(* Logix 5000 project; controller reports 1756-L63 rev 20.11; software revision 20.04; part 47 of 52 *)

        [152].log_data[58].time := 3600.0, [152].log_data[58].valid := 1, [152].log_data[59].time := 3600.0, [152].log_data[59].valid := 1, [152].log_data[60].valid := 1, [152].log_data[61].valid := 1, [152].log_data[62].valid := 1, [152].log_data[63].valid := 1, [152].log_data[64].valid := 1, [152].log_data[65].valid := 1, [152].log_data[66].valid := 1, [152].log_data[67].valid := 1, [152].log_data[68].valid := 1, [152].log_data[69].valid := 1, [152].log_data[70].valid := 1, [152].log_data[71].valid := 1, [152].log_data[72].valid := 1, [152].log_data[73].valid := 1, [152].log_data[74].valid := 1, [152].log_data[75].valid := 1, [152].log_data[76].valid := 1, [152].log_data[77].valid := 1, [152].log_data[78].valid := 1, [152].log_data[79].valid := 1, [152].log_data[80].valid := 1, [152].log_data[81].valid := 1, [152].log_data[82].valid := 1, [152].log_data[83].valid := 1, [152].log_data[84].valid := 1, [152].log_data[85].valid := 1, [152].log_data[86].valid := 1, [152].log_data[87].valid := 1, [152].log_data[88].valid := 1, [152].log_data[89].valid := 1, [152].log_data[90].valid := 1, [152].log_data[91].valid := 1, [152].log_data[92].valid := 1, [152].log_data[93].valid := 1, [152].log_data[94].valid := 1, [152].log_data[95].valid := 1, [152].log_data[96].valid := 1, [152].log_data[97].valid := 1, [152].log_data[98].valid := 1, [152].log_data[99].valid := 1, [152].log_data[100].valid := 1, [152].log_data[101].valid := 1, [152].log_data[102].valid := 1, [152].log_data[103].valid := 1, [152].log_data[104].valid := 1, [152].log_data[105].valid := 1, [152].log_data[106].valid := 1, [152].log_data[107].valid := 1, [152].log_data[108].valid := 1, [152].log_data[109].valid := 1, [152].log_data[110].valid := 1, [152].log_data[111].valid := 1, [152].log_data[112].valid := 1, [152].log_data[113].valid := 1, [152].log_data[114].valid := 1, [152].log_data[115].valid := 1,
        [152].log_data[116].valid := 1, [152].log_data[117].valid := 1, [152].log_data[118].valid := 1, [152].log_data[119].valid := 1, [152].log_data[120].valid := 1, [152].log_data[121].valid := 1, [152].log_data[122].valid := 1, [152].log_data[123].valid := 1, [152].log_data[124].valid := 1, [152].time.Year := 2023, [152].time.Month := 1, [152].time.Day := 19, [152].time.Hour := 11, [152].time.Minute := 59, [152].time.Second := 59, [153].log_data[0].min := 1.0, [153].log_data[0].max := 1.0, [153].log_data[0].total := 3600.0, [153].log_data[0].time := 3600.0, [153].log_data[0].valid := 1, [153].log_data[1].time := 3600.0, [153].log_data[1].valid := 1, [153].log_data[2].time := 3600.0, [153].log_data[2].valid := 1, [153].log_data[3].time := 3600.0, [153].log_data[3].valid := 1, [153].log_data[4].time := 3600.0, [153].log_data[4].valid := 1, [153].log_data[5].time := 3600.0, [153].log_data[5].valid := 1, [153].log_data[6].time := 3600.0, [153].log_data[6].valid := 1, [153].log_data[7].time := 3600.0, [153].log_data[7].valid := 1, [153].log_data[8].min := 1.0, [153].log_data[8].max := 1.0, [153].log_data[8].total := 3600.0, [153].log_data[8].time := 3600.0, [153].log_data[8].valid := 1, [153].log_data[9].min := 1.0, [153].log_data[9].max := 1.0, [153].log_data[9].total := 3600.0, [153].log_data[9].time := 3600.0, [153].log_data[9].valid := 1, [153].log_data[10].min := 1.0, [153].log_data[10].max := 1.0, [153].log_data[10].total := 3600.0, [153].log_data[10].time := 3600.0, [153].log_data[10].valid := 1, [153].log_data[11].time := 3600.0, [153].log_data[11].valid := 1, [153].log_data[12].min := 1.0, [153].log_data[12].max := 1.0, [153].log_data[12].total := 3600.0, [153].log_data[12].time := 3600.0, [153].log_data[12].valid := 1, [153].log_data[13].min := 1.0, [153].log_data[13].max := 1.0, [153].log_data[13].total := 3600.0, [153].log_data[13].time := 3600.0,
        [153].log_data[13].valid := 1, [153].log_data[14].time := 3600.0, [153].log_data[14].valid := 1, [153].log_data[15].time := 3600.0, [153].log_data[15].valid := 1, [153].log_data[16].time := 3600.0, [153].log_data[16].valid := 1, [153].log_data[17].min := 1.0, [153].log_data[17].max := 1.0, [153].log_data[17].total := 3600.0, [153].log_data[17].time := 3600.0, [153].log_data[17].valid := 1, [153].log_data[18].time := 3600.0, [153].log_data[18].valid := 1, [153].log_data[19].time := 3600.0, [153].log_data[19].valid := 1, [153].log_data[20].time := 3600.0, [153].log_data[20].valid := 1, [153].log_data[21].min := 1.0, [153].log_data[21].max := 1.0, [153].log_data[21].total := 3600.0, [153].log_data[21].time := 3600.0, [153].log_data[21].valid := 1, [153].log_data[22].time := 3600.0, [153].log_data[22].valid := 1, [153].log_data[23].time := 3600.0, [153].log_data[23].valid := 1, [153].log_data[24].time := 3600.0, [153].log_data[24].valid := 1, [153].log_data[25].time := 3600.0, [153].log_data[25].valid := 1, [153].log_data[26].time := 3600.0, [153].log_data[26].valid := 1, [153].log_data[27].time := 3600.0, [153].log_data[27].valid := 1, [153].log_data[28].time := 3600.0, [153].log_data[28].valid := 1, [153].log_data[29].min := 1.0, [153].log_data[29].max := 1.0, [153].log_data[29].total := 3600.0, [153].log_data[29].time := 3600.0, [153].log_data[29].valid := 1, [153].log_data[30].min := 1.0, [153].log_data[30].max := 1.0, [153].log_data[30].total := 3600.0, [153].log_data[30].time := 3600.0, [153].log_data[30].valid := 1, [153].log_data[31].max := 1.0, [153].log_data[31].total := 1629.749, [153].log_data[31].time := 3600.0, [153].log_data[31].valid := 1, [153].log_data[32].max := 1.0, [153].log_data[32].total := 1481.7471, [153].log_data[32].time := 3600.0, [153].log_data[32].maxminute := 11, [153].log_data[32].valid := 1, [153].log_data[33].time := 3600.0, [153].log_data[33].valid := 1, [153].log_data[34].time := 3600.0, [153].log_data[34].valid := 1,
        [153].log_data[35].max := 1.0, [153].log_data[35].total := 1629.998, [153].log_data[35].time := 3600.0, [153].log_data[35].maxminute := 8, [153].log_data[35].valid := 1, [153].log_data[36].max := 1.0, [153].log_data[36].total := 1480.249, [153].log_data[36].time := 3600.0, [153].log_data[36].minminute := 6, [153].log_data[36].valid := 1, [153].log_data[37].time := 3600.0, [153].log_data[37].valid := 1, [153].log_data[38].time := 3600.0, [153].log_data[38].valid := 1, [153].log_data[39].min := 0.9945885, [153].log_data[39].max := 1.0051882, [153].log_data[39].total := 3601.9607, [153].log_data[39].time := 3600.0, [153].log_data[39].minminute := 59, [153].log_data[39].maxminute := 44, [153].log_data[39].valid := 1, [153].log_data[40].min := 7.5950956, [153].log_data[40].max := 7.6195536, [153].log_data[40].total := 27406.98, [153].log_data[40].time := 3600.0, [153].log_data[40].minminute := 52, [153].log_data[40].maxminute := 59, [153].log_data[40].valid := 1, [153].log_data[41].min := 0.021362305, [153].log_data[41].max := 0.023521485, [153].log_data[41].total := 80.782776, [153].log_data[41].time := 3600.0, [153].log_data[41].minminute := 25, [153].log_data[41].maxminute := 24, [153].log_data[41].valid := 1, [153].log_data[42].min := 2.290936, [153].log_data[42].max := 2.296236, [153].log_data[42].total := 8256.996, [153].log_data[42].time := 3600.0, [153].log_data[42].minminute := 43, [153].log_data[42].maxminute := 14, [153].log_data[42].valid := 1, [153].log_data[43].min := -0.27999878, [153].log_data[43].max := -0.22000122, [153].log_data[43].total := -891.35376, [153].log_data[43].time := 3600.0, [153].log_data[43].maxminute := 45, [153].log_data[43].valid := 1, [153].log_data[44].min := -0.30000305, [153].log_data[44].max := -0.26000214, [153].log_data[44].total := -1000.0248, [153].log_data[44].time := 3600.0, [153].log_data[44].maxminute := 35, [153].log_data[44].valid := 1, [153].log_data[45].time := 3600.0, [153].log_data[45].valid := 1, [153].log_data[46].time := 3600.0, [153].log_data[46].valid := 1, [153].log_data[47].time := 3600.0, [153].log_data[47].valid := 1,
        [153].log_data[48].min := 6.567313, [153].log_data[48].max := 6.784686, [153].log_data[48].total := 24147.303, [153].log_data[48].time := 3600.0, [153].log_data[48].minminute := 14, [153].log_data[48].maxminute := 29, [153].log_data[48].valid := 1, [153].log_data[49].min := 6.8652577, [153].log_data[49].max := 9.493403, [153].log_data[49].total := 29615.246, [153].log_data[49].time := 3600.0, [153].log_data[49].minminute := 15, [153].log_data[49].maxminute := 59, [153].log_data[49].valid := 1, [153].log_data[50].min := 2.0285335, [153].log_data[50].max := 2.1149805, [153].log_data[50].total := 7461.926, [153].log_data[50].time := 3600.0, [153].log_data[50].minminute := 58, [153].log_data[50].valid := 1, [153].log_data[51].time := 3600.0, [153].log_data[51].valid := 1, [153].log_data[52].min := -2.7600021, [153].log_data[52].max := 0.13999939, [153].log_data[52].total := -7610.8003, [153].log_data[52].time := 3600.0, [153].log_data[52].minminute := 21, [153].log_data[52].maxminute := 31, [153].log_data[52].valid := 1, [153].log_data[53].min := -2.5, [153].log_data[53].max := 0.27999878, [153].log_data[53].total := -7005.6523, [153].log_data[53].time := 3600.0, [153].log_data[53].minminute := 50, [153].log_data[53].maxminute := 7, [153].log_data[53].valid := 1, [153].log_data[54].max := 0.5255, [153].log_data[54].total := 1233.0619, [153].log_data[54].time := 3600.0, [153].log_data[54].valid := 1, [153].log_data[55].max := 0.55300003, [153].log_data[55].total := 1235.2316, [153].log_data[55].time := 3600.0, [153].log_data[55].minminute := 6, [153].log_data[55].maxminute := 50, [153].log_data[55].valid := 1, [153].log_data[56].min := 0.15895009, [153].log_data[56].max := 0.15946046, [153].log_data[56].total := 573.08417, [153].log_data[56].time := 3600.0, [153].log_data[56].minminute := 2, [153].log_data[56].maxminute := 44, [153].log_data[56].valid := 1, [153].log_data[57].min := 0.18721606, [153].log_data[57].max := 0.18976782, [153].log_data[57].total := 676.8789, [153].log_data[57].time := 3600.0, [153].log_data[57].minminute := 24, [153].log_data[57].maxminute := 6, [153].log_data[57].valid := 1,
        [153].log_data[58].time := 3600.0, [153].log_data[58].valid := 1, [153].log_data[59].time := 3600.0, [153].log_data[59].valid := 1, [153].log_data[60].valid := 1, [153].log_data[61].valid := 1, [153].log_data[62].valid := 1, [153].log_data[63].valid := 1, [153].log_data[64].valid := 1, [153].log_data[65].valid := 1, [153].log_data[66].valid := 1, [153].log_data[67].valid := 1, [153].log_data[68].valid := 1, [153].log_data[69].valid := 1, [153].log_data[70].valid := 1, [153].log_data[71].valid := 1, [153].log_data[72].valid := 1, [153].log_data[73].valid := 1, [153].log_data[74].valid := 1, [153].log_data[75].valid := 1, [153].log_data[76].valid := 1, [153].log_data[77].valid := 1, [153].log_data[78].valid := 1, [153].log_data[79].valid := 1, [153].log_data[80].valid := 1, [153].log_data[81].valid := 1, [153].log_data[82].valid := 1, [153].log_data[83].valid := 1, [153].log_data[84].valid := 1, [153].log_data[85].valid := 1, [153].log_data[86].valid := 1, [153].log_data[87].valid := 1, [153].log_data[88].valid := 1, [153].log_data[89].valid := 1, [153].log_data[90].valid := 1, [153].log_data[91].valid := 1, [153].log_data[92].valid := 1, [153].log_data[93].valid := 1, [153].log_data[94].valid := 1, [153].log_data[95].valid := 1, [153].log_data[96].valid := 1, [153].log_data[97].valid := 1, [153].log_data[98].valid := 1, [153].log_data[99].valid := 1, [153].log_data[100].valid := 1, [153].log_data[101].valid := 1, [153].log_data[102].valid := 1, [153].log_data[103].valid := 1, [153].log_data[104].valid := 1, [153].log_data[105].valid := 1, [153].log_data[106].valid := 1, [153].log_data[107].valid := 1, [153].log_data[108].valid := 1, [153].log_data[109].valid := 1, [153].log_data[110].valid := 1, [153].log_data[111].valid := 1, [153].log_data[112].valid := 1, [153].log_data[113].valid := 1, [153].log_data[114].valid := 1, [153].log_data[115].valid := 1,
        [153].log_data[116].valid := 1, [153].log_data[117].valid := 1, [153].log_data[118].valid := 1, [153].log_data[119].valid := 1, [153].log_data[120].valid := 1, [153].log_data[121].valid := 1, [153].log_data[122].valid := 1, [153].log_data[123].valid := 1, [153].log_data[124].valid := 1, [153].time.Year := 2023, [153].time.Month := 1, [153].time.Day := 19, [153].time.Hour := 12, [153].time.Minute := 59, [153].time.Second := 59, [154].log_data[0].min := 1.0, [154].log_data[0].max := 1.0, [154].log_data[0].total := 3600.0, [154].log_data[0].time := 3600.0, [154].log_data[0].valid := 1, [154].log_data[1].max := 1.0, [154].log_data[1].total := 541.0, [154].log_data[1].time := 3600.0, [154].log_data[1].maxminute := 16, [154].log_data[1].valid := 1, [154].log_data[2].max := 1.0, [154].log_data[2].total := 537.5, [154].log_data[2].time := 3600.0, [154].log_data[2].maxminute := 16, [154].log_data[2].valid := 1, [154].log_data[3].time := 3600.0, [154].log_data[3].valid := 1, [154].log_data[4].time := 3600.0, [154].log_data[4].valid := 1, [154].log_data[5].max := 1.0, [154].log_data[5].total := 234.0, [154].log_data[5].time := 3600.0, [154].log_data[5].maxminute := 18, [154].log_data[5].valid := 1, [154].log_data[6].time := 3600.0, [154].log_data[6].valid := 1, [154].log_data[7].time := 3600.0, [154].log_data[7].valid := 1, [154].log_data[8].min := 1.0, [154].log_data[8].max := 1.0, [154].log_data[8].total := 3600.0, [154].log_data[8].time := 3600.0, [154].log_data[8].valid := 1, [154].log_data[9].min := 1.0, [154].log_data[9].max := 1.0, [154].log_data[9].total := 3600.0, [154].log_data[9].time := 3600.0, [154].log_data[9].valid := 1, [154].log_data[10].min := 1.0, [154].log_data[10].max := 1.0, [154].log_data[10].total := 3600.0, [154].log_data[10].time := 3600.0, [154].log_data[10].valid := 1, [154].log_data[11].time := 3600.0, [154].log_data[11].valid := 1,
        [154].log_data[12].min := 1.0, [154].log_data[12].max := 1.0, [154].log_data[12].total := 3600.0, [154].log_data[12].time := 3600.0, [154].log_data[12].valid := 1, [154].log_data[13].min := 1.0, [154].log_data[13].max := 1.0, [154].log_data[13].total := 3600.0, [154].log_data[13].time := 3600.0, [154].log_data[13].valid := 1, [154].log_data[14].time := 3600.0, [154].log_data[14].valid := 1, [154].log_data[15].time := 3600.0, [154].log_data[15].valid := 1, [154].log_data[16].time := 3600.0, [154].log_data[16].valid := 1, [154].log_data[17].min := 1.0, [154].log_data[17].max := 1.0, [154].log_data[17].total := 3600.0, [154].log_data[17].time := 3600.0, [154].log_data[17].valid := 1, [154].log_data[18].time := 3600.0, [154].log_data[18].valid := 1, [154].log_data[19].time := 3600.0, [154].log_data[19].valid := 1, [154].log_data[20].time := 3600.0, [154].log_data[20].valid := 1, [154].log_data[21].min := 1.0, [154].log_data[21].max := 1.0, [154].log_data[21].total := 3600.0, [154].log_data[21].time := 3600.0, [154].log_data[21].valid := 1, [154].log_data[22].time := 3600.0, [154].log_data[22].valid := 1, [154].log_data[23].time := 3600.0, [154].log_data[23].valid := 1, [154].log_data[24].time := 3600.0, [154].log_data[24].valid := 1, [154].log_data[25].time := 3600.0, [154].log_data[25].valid := 1, [154].log_data[26].time := 3600.0, [154].log_data[26].valid := 1, [154].log_data[27].time := 3600.0, [154].log_data[27].valid := 1, [154].log_data[28].time := 3600.0, [154].log_data[28].valid := 1, [154].log_data[29].min := 1.0, [154].log_data[29].max := 1.0, [154].log_data[29].total := 3600.0, [154].log_data[29].time := 3600.0, [154].log_data[29].valid := 1, [154].log_data[30].min := 1.0, [154].log_data[30].max := 1.0, [154].log_data[30].total := 3600.0, [154].log_data[30].time := 3600.0, [154].log_data[30].valid := 1, [154].log_data[31].max := 1.0, [154].log_data[31].total := 1629.998, [154].log_data[31].time := 3600.0, [154].log_data[31].maxminute := 3,
        [154].log_data[31].valid := 1, [154].log_data[32].max := 1.0, [154].log_data[32].total := 1440.998, [154].log_data[32].time := 3600.0, [154].log_data[32].minminute := 2, [154].log_data[32].valid := 1, [154].log_data[33].time := 3600.0, [154].log_data[33].valid := 1, [154].log_data[34].time := 3600.0, [154].log_data[34].valid := 1, [154].log_data[35].max := 1.0, [154].log_data[35].total := 1489.7471, [154].log_data[35].time := 3600.0, [154].log_data[35].maxminute := 11, [154].log_data[35].valid := 1, [154].log_data[36].max := 1.0, [154].log_data[36].total := 1629.998, [154].log_data[36].time := 3600.0, [154].log_data[36].valid := 1, [154].log_data[37].max := 7.485309, [154].log_data[37].total := 3503.0806, [154].log_data[37].time := 3600.0, [154].log_data[37].maxminute := 16, [154].log_data[37].valid := 1, [154].log_data[38].time := 3600.0, [154].log_data[38].valid := 1, [154].log_data[39].min := 0.9944707, [154].log_data[39].max := 1.0215589, [154].log_data[39].total := 3606.9067, [154].log_data[39].time := 3600.0, [154].log_data[39].minminute := 3, [154].log_data[39].maxminute := 23, [154].log_data[39].valid := 1, [154].log_data[40].min := 7.6019654, [154].log_data[40].max := 7.6297207, [154].log_data[40].total := 27414.703, [154].log_data[40].time := 3600.0, [154].log_data[40].minminute := 13, [154].log_data[40].maxminute := 6, [154].log_data[40].valid := 1, [154].log_data[41].min := 0.021754883, [154].log_data[41].max := 0.022540038, [154].log_data[41].total := 79.7362, [154].log_data[41].time := 3600.0, [154].log_data[41].minminute := 48, [154].log_data[41].valid := 1, [154].log_data[42].min := 2.2910538, [154].log_data[42].max := 2.296236, [154].log_data[42].total := 8256.574, [154].log_data[42].time := 3600.0, [154].log_data[42].minminute := 54, [154].log_data[42].maxminute := 22, [154].log_data[42].valid := 1, [154].log_data[43].min := -0.23999786, [154].log_data[43].max := -0.19999695, [154].log_data[43].total := -764.9952, [154].log_data[43].time := 3600.0, [154].log_data[43].maxminute := 26, [154].log_data[43].valid := 1, [154].log_data[44].min := -0.27999878,
        [154].log_data[44].max := -0.22000122, [154].log_data[44].total := -872.0464, [154].log_data[44].time := 3600.0, [154].log_data[44].minminute := 7, [154].log_data[44].maxminute := 39, [154].log_data[44].valid := 1, [154].log_data[45].time := 3600.0, [154].log_data[45].valid := 1, [154].log_data[46].time := 3600.0, [154].log_data[46].valid := 1, [154].log_data[47].time := 3600.0, [154].log_data[47].valid := 1, [154].log_data[48].min := 6.576932, [154].log_data[48].max := 6.9325333, [154].log_data[48].total := 24178.086, [154].log_data[48].time := 3600.0, [154].log_data[48].minminute := 47, [154].log_data[48].maxminute := 21, [154].log_data[48].valid := 1, [154].log_data[49].min := 6.850929, [154].log_data[49].max := 9.543064, [154].log_data[49].total := 29634.871, [154].log_data[49].time := 3600.0, [154].log_data[49].minminute := 44, [154].log_data[49].maxminute := 9, [154].log_data[49].valid := 1, [154].log_data[50].min := 2.0040364, [154].log_data[50].max := 2.1119182, [154].log_data[50].total := 7430.037, [154].log_data[50].time := 3600.0, [154].log_data[50].minminute := 18, [154].log_data[50].maxminute := 25, [154].log_data[50].valid := 1, [154].log_data[51].time := 3600.0, [154].log_data[51].valid := 1, [154].log_data[52].min := -2.8600006, [154].log_data[52].max := 0.16000366, [154].log_data[52].total := -7486.2666, [154].log_data[52].time := 3600.0, [154].log_data[52].minminute := 4, [154].log_data[52].maxminute := 34, [154].log_data[52].valid := 1, [154].log_data[53].min := -2.5, [154].log_data[53].max := 0.16000366, [154].log_data[53].total := -7109.941, [154].log_data[53].time := 3600.0, [154].log_data[53].minminute := 12, [154].log_data[53].maxminute := 21, [154].log_data[53].valid := 1, [154].log_data[54].max := 0.537, [154].log_data[54].total := 1217.782, [154].log_data[54].time := 3600.0, [154].log_data[54].minminute := 2, [154].log_data[54].maxminute := 46, [154].log_data[54].valid := 1, [154].log_data[55].max := 0.5395, [154].log_data[55].total := 1236.7081, [154].log_data[55].time := 3600.0, [154].log_data[55].maxminute := 32, [154].log_data[55].valid := 1,
        [154].log_data[56].min := 0.15902862, [154].log_data[56].max := 0.15946046, [154].log_data[56].total := 573.1385, [154].log_data[56].time := 3600.0, [154].log_data[56].minminute := 47, [154].log_data[56].maxminute := 1, [154].log_data[56].valid := 1, [154].log_data[57].min := 0.18595977, [154].log_data[57].max := 0.18815826, [154].log_data[57].total := 674.85864, [154].log_data[57].time := 3600.0, [154].log_data[57].minminute := 54, [154].log_data[57].maxminute := 40, [154].log_data[57].valid := 1, [154].log_data[58].time := 3600.0, [154].log_data[58].valid := 1, [154].log_data[59].time := 3600.0, [154].log_data[59].valid := 1, [154].log_data[60].time := 652.249, [154].log_data[60].minminute := 49, [154].log_data[60].maxminute := 49, [154].log_data[60].valid := 1, [154].log_data[61].valid := 1, [154].log_data[62].valid := 1, [154].log_data[63].valid := 1, [154].log_data[64].valid := 1, [154].log_data[65].valid := 1, [154].log_data[66].valid := 1, [154].log_data[67].valid := 1, [154].log_data[68].valid := 1, [154].log_data[69].valid := 1, [154].log_data[70].valid := 1, [154].log_data[71].valid := 1, [154].log_data[72].valid := 1, [154].log_data[73].valid := 1, [154].log_data[74].valid := 1, [154].log_data[75].valid := 1, [154].log_data[76].valid := 1, [154].log_data[77].valid := 1, [154].log_data[78].valid := 1, [154].log_data[79].valid := 1, [154].log_data[80].valid := 1, [154].log_data[81].valid := 1, [154].log_data[82].valid := 1, [154].log_data[83].valid := 1, [154].log_data[84].valid := 1, [154].log_data[85].valid := 1, [154].log_data[86].valid := 1, [154].log_data[87].valid := 1, [154].log_data[88].valid := 1, [154].log_data[89].valid := 1, [154].log_data[90].valid := 1, [154].log_data[91].valid := 1, [154].log_data[92].valid := 1, [154].log_data[93].valid := 1, [154].log_data[94].valid := 1, [154].log_data[95].valid := 1, [154].log_data[96].valid := 1, [154].log_data[97].valid := 1, [154].log_data[98].valid := 1,
        [154].log_data[99].valid := 1, [154].log_data[100].valid := 1, [154].log_data[101].valid := 1, [154].log_data[102].valid := 1, [154].log_data[103].valid := 1, [154].log_data[104].valid := 1, [154].log_data[105].valid := 1, [154].log_data[106].valid := 1, [154].log_data[107].valid := 1, [154].log_data[108].valid := 1, [154].log_data[109].valid := 1, [154].log_data[110].valid := 1, [154].log_data[111].valid := 1, [154].log_data[112].valid := 1, [154].log_data[113].valid := 1, [154].log_data[114].valid := 1, [154].log_data[115].valid := 1, [154].log_data[116].valid := 1, [154].log_data[117].valid := 1, [154].log_data[118].valid := 1, [154].log_data[119].valid := 1, [154].log_data[120].valid := 1, [154].log_data[121].valid := 1, [154].log_data[122].valid := 1, [154].log_data[123].valid := 1, [154].log_data[124].valid := 1, [154].time.Year := 2023, [154].time.Month := 1, [154].time.Day := 19, [154].time.Hour := 13, [154].time.Minute := 59, [154].time.Second := 59, [155].log_data[0].min := 1.0, [155].log_data[0].max := 1.0, [155].log_data[0].total := 3600.0, [155].log_data[0].time := 3600.0, [155].log_data[0].valid := 1, [155].log_data[1].time := 3600.0, [155].log_data[1].valid := 1, [155].log_data[2].time := 3600.0, [155].log_data[2].valid := 1, [155].log_data[3].time := 3600.0, [155].log_data[3].valid := 1, [155].log_data[4].time := 3600.0, [155].log_data[4].valid := 1, [155].log_data[5].time := 3600.0, [155].log_data[5].valid := 1, [155].log_data[6].time := 3600.0, [155].log_data[6].valid := 1, [155].log_data[7].time := 3600.0, [155].log_data[7].valid := 1, [155].log_data[8].max := 1.0, [155].log_data[8].total := 2888.251, [155].log_data[8].time := 3600.0, [155].log_data[8].minminute := 48, [155].log_data[8].valid := 1, [155].log_data[9].max := 1.0, [155].log_data[9].total := 2888.251, [155].log_data[9].time := 3600.0, [155].log_data[9].minminute := 48,
        [155].log_data[9].valid := 1, [155].log_data[10].min := 1.0, [155].log_data[10].max := 1.0, [155].log_data[10].total := 3600.0, [155].log_data[10].time := 3600.0, [155].log_data[10].valid := 1, [155].log_data[11].time := 3600.0, [155].log_data[11].valid := 1, [155].log_data[12].min := 1.0, [155].log_data[12].max := 1.0, [155].log_data[12].total := 3600.0, [155].log_data[12].time := 3600.0, [155].log_data[12].valid := 1, [155].log_data[13].min := 1.0, [155].log_data[13].max := 1.0, [155].log_data[13].total := 3600.0, [155].log_data[13].time := 3600.0, [155].log_data[13].valid := 1, [155].log_data[14].time := 3600.0, [155].log_data[14].valid := 1, [155].log_data[15].time := 3600.0, [155].log_data[15].valid := 1, [155].log_data[16].time := 3600.0, [155].log_data[16].valid := 1, [155].log_data[17].min := 1.0, [155].log_data[17].max := 1.0, [155].log_data[17].total := 3600.0, [155].log_data[17].time := 3600.0, [155].log_data[17].valid := 1, [155].log_data[18].max := 1.0, [155].log_data[18].total := 144.249, [155].log_data[18].time := 3600.0, [155].log_data[18].maxminute := 55, [155].log_data[18].valid := 1, [155].log_data[19].max := 1.0, [155].log_data[19].total := 30.5, [155].log_data[19].time := 3600.0, [155].log_data[19].maxminute := 56, [155].log_data[19].valid := 1, [155].log_data[20].time := 3600.0, [155].log_data[20].valid := 1, [155].log_data[21].min := 1.0, [155].log_data[21].max := 1.0, [155].log_data[21].total := 3600.0, [155].log_data[21].time := 3600.0, [155].log_data[21].valid := 1, [155].log_data[22].time := 3600.0, [155].log_data[22].valid := 1, [155].log_data[23].time := 3600.0, [155].log_data[23].valid := 1, [155].log_data[24].time := 3600.0, [155].log_data[24].valid := 1, [155].log_data[25].time := 3600.0, [155].log_data[25].valid := 1, [155].log_data[26].time := 3600.0, [155].log_data[26].valid := 1, [155].log_data[27].time := 3600.0, [155].log_data[27].valid := 1, [155].log_data[28].time := 3600.0, [155].log_data[28].valid := 1,
        [155].log_data[29].min := 1.0, [155].log_data[29].max := 1.0, [155].log_data[29].total := 3600.0, [155].log_data[29].time := 3600.0, [155].log_data[29].valid := 1, [155].log_data[30].min := 1.0, [155].log_data[30].max := 1.0, [155].log_data[30].total := 3600.0, [155].log_data[30].time := 3600.0, [155].log_data[30].valid := 1, [155].log_data[31].max := 1.0, [155].log_data[31].total := 1086.498, [155].log_data[31].time := 3600.0, [155].log_data[31].maxminute := 7, [155].log_data[31].valid := 1, [155].log_data[32].max := 1.0, [155].log_data[32].total := 1423.749, [155].log_data[32].time := 3600.0, [155].log_data[32].minminute := 5, [155].log_data[32].valid := 1, [155].log_data[33].time := 3600.0, [155].log_data[33].valid := 1, [155].log_data[34].time := 3600.0, [155].log_data[34].valid := 1, [155].log_data[35].max := 1.0, [155].log_data[35].total := 1226.498, [155].log_data[35].time := 3600.0, [155].log_data[35].minminute := 2, [155].log_data[35].valid := 1, [155].log_data[36].max := 1.0, [155].log_data[36].total := 1224.2471, [155].log_data[36].time := 3600.0, [155].log_data[36].maxminute := 3, [155].log_data[36].valid := 1, [155].log_data[37].time := 3600.0, [155].log_data[37].valid := 1, [155].log_data[38].time := 3600.0, [155].log_data[38].valid := 1, [155].log_data[39].min := 0.99423516, [155].log_data[39].max := 1.0055416, [155].log_data[39].total := 3603.8801, [155].log_data[39].time := 3600.0, [155].log_data[39].minminute := 18, [155].log_data[39].maxminute := 12, [155].log_data[39].valid := 1, [155].log_data[40].min := 7.5989423, [155].log_data[40].max := 7.6195536, [155].log_data[40].total := 27415.486, [155].log_data[40].time := 3600.0, [155].log_data[40].minminute := 57, [155].log_data[40].maxminute := 5, [155].log_data[40].valid := 1, [155].log_data[41].min := 0.021362305, [155].log_data[41].max := 0.022540038, [155].log_data[41].total := 79.09212, [155].log_data[41].time := 3600.0, [155].log_data[41].minminute := 24, [155].log_data[41].maxminute := 24, [155].log_data[41].valid := 1, [155].log_data[42].min := 2.290936,
        [155].log_data[42].max := 2.2957647, [155].log_data[42].total := 8256.586, [155].log_data[42].time := 3600.0, [155].log_data[42].minminute := 1, [155].log_data[42].maxminute := 11, [155].log_data[42].valid := 1, [155].log_data[43].min := -0.19999695, [155].log_data[43].max := -0.19999695, [155].log_data[43].total := -719.9707, [155].log_data[43].time := 3600.0, [155].log_data[43].valid := 1, [155].log_data[44].min := -0.30000305, [155].log_data[44].max := -0.22000122, [155].log_data[44].total := -796.0592, [155].log_data[44].time := 3600.0, [155].log_data[44].minminute := 58, [155].log_data[44].valid := 1, [155].log_data[45].time := 3600.0, [155].log_data[45].valid := 1, [155].log_data[46].time := 3600.0, [155].log_data[46].valid := 1, [155].log_data[47].time := 3600.0, [155].log_data[47].valid := 1, [155].log_data[48].min := 6.7365947, [155].log_data[48].max := 6.7885337, [155].log_data[48].total := 24300.299, [155].log_data[48].time := 3600.0, [155].log_data[48].minminute := 50, [155].log_data[48].maxminute := 1, [155].log_data[48].valid := 1, [155].log_data[49].min := 8.224183, [155].log_data[49].max := 9.507536, [155].log_data[49].total := 33398.145, [155].log_data[49].time := 3600.0, [155].log_data[49].maxminute := 56, [155].log_data[49].valid := 1, [155].log_data[50].min := 1.9989722, [155].log_data[50].max := 2.1001406, [155].log_data[50].total := 7358.492, [155].log_data[50].time := 3600.0, [155].log_data[50].minminute := 48, [155].log_data[50].maxminute := 59, [155].log_data[50].valid := 1, [155].log_data[51].time := 3600.0, [155].log_data[51].valid := 1, [155].log_data[52].min := -2.8600006, [155].log_data[52].max := 0.16000366, [155].log_data[52].total := -6845.63, [155].log_data[52].time := 3600.0, [155].log_data[52].minminute := 28, [155].log_data[52].maxminute := 5, [155].log_data[52].valid := 1, [155].log_data[53].min := -2.5200043, [155].log_data[53].max := 0.16000366, [155].log_data[53].total := -6421.268, [155].log_data[53].time := 3600.0, [155].log_data[53].minminute := 16, [155].log_data[53].maxminute := 3, [155].log_data[53].valid := 1, [155].log_data[54].max := 0.564,
        [155].log_data[54].total := 996.96844, [155].log_data[54].time := 3600.0, [155].log_data[54].minminute := 5, [155].log_data[54].maxminute := 28, [155].log_data[54].valid := 1, [155].log_data[55].max := 0.51350003, [155].log_data[55].total := 971.1236, [155].log_data[55].time := 3600.0, [155].log_data[55].minminute := 2, [155].log_data[55].maxminute := 35, [155].log_data[55].valid := 1, [155].log_data[56].min := 0.15898935, [155].log_data[56].max := 0.15938194, [155].log_data[56].total := 572.8917, [155].log_data[56].time := 3600.0, [155].log_data[56].minminute := 38, [155].log_data[56].valid := 1, [155].log_data[57].min := 0.18599902, [155].log_data[57].max := 0.18658794, [155].log_data[57].total := 670.5091, [155].log_data[57].time := 3600.0, [155].log_data[57].maxminute := 50, [155].log_data[57].valid := 1, [155].log_data[58].time := 3600.0, [155].log_data[58].valid := 1, [155].log_data[59].time := 3600.0, [155].log_data[59].valid := 1, [155].log_data[60].time := 3600.0, [155].log_data[60].valid := 1, [155].log_data[61].valid := 1, [155].log_data[62].valid := 1, [155].log_data[63].valid := 1, [155].log_data[64].valid := 1, [155].log_data[65].valid := 1, [155].log_data[66].valid := 1, [155].log_data[67].valid := 1, [155].log_data[68].valid := 1, [155].log_data[69].valid := 1, [155].log_data[70].valid := 1, [155].log_data[71].valid := 1, [155].log_data[72].valid := 1, [155].log_data[73].valid := 1, [155].log_data[74].valid := 1, [155].log_data[75].valid := 1, [155].log_data[76].valid := 1, [155].log_data[77].valid := 1, [155].log_data[78].valid := 1, [155].log_data[79].valid := 1, [155].log_data[80].valid := 1, [155].log_data[81].valid := 1, [155].log_data[82].valid := 1, [155].log_data[83].valid := 1, [155].log_data[84].valid := 1, [155].log_data[85].valid := 1, [155].log_data[86].valid := 1, [155].log_data[87].valid := 1, [155].log_data[88].valid := 1, [155].log_data[89].valid := 1, [155].log_data[90].valid := 1, [155].log_data[91].valid := 1,
        [155].log_data[92].valid := 1, [155].log_data[93].valid := 1, [155].log_data[94].valid := 1, [155].log_data[95].valid := 1, [155].log_data[96].valid := 1, [155].log_data[97].valid := 1, [155].log_data[98].valid := 1, [155].log_data[99].valid := 1, [155].log_data[100].valid := 1, [155].log_data[101].valid := 1, [155].log_data[102].valid := 1, [155].log_data[103].valid := 1, [155].log_data[104].valid := 1, [155].log_data[105].valid := 1, [155].log_data[106].valid := 1, [155].log_data[107].valid := 1, [155].log_data[108].valid := 1, [155].log_data[109].valid := 1, [155].log_data[110].valid := 1, [155].log_data[111].valid := 1, [155].log_data[112].valid := 1, [155].log_data[113].valid := 1, [155].log_data[114].valid := 1, [155].log_data[115].valid := 1, [155].log_data[116].valid := 1, [155].log_data[117].valid := 1, [155].log_data[118].valid := 1, [155].log_data[119].valid := 1, [155].log_data[120].valid := 1, [155].log_data[121].valid := 1, [155].log_data[122].valid := 1, [155].log_data[123].valid := 1, [155].log_data[124].valid := 1, [155].time.Year := 2023, [155].time.Month := 1, [155].time.Day := 19, [155].time.Hour := 14, [155].time.Minute := 59, [155].time.Second := 59, [156].log_data[0].min := 1.0, [156].log_data[0].max := 1.0, [156].log_data[0].total := 1572.0, [156].log_data[0].time := 1572.0, [156].log_data[0].valid := 1, [156].log_data[1].max := 1.0, [156].log_data[1].total := 143.749, [156].log_data[1].time := 1572.0, [156].log_data[1].maxminute := 23, [156].log_data[1].valid := 1, [156].log_data[2].max := 1.0, [156].log_data[2].total := 140.249, [156].log_data[2].time := 1572.0, [156].log_data[2].maxminute := 23, [156].log_data[2].valid := 1, [156].log_data[3].time := 1572.0, [156].log_data[3].valid := 1, [156].log_data[4].time := 1572.0, [156].log_data[4].valid := 1, [156].log_data[5].time := 1572.0, [156].log_data[5].valid := 1,
        [156].log_data[6].time := 1572.0, [156].log_data[6].valid := 1, [156].log_data[7].time := 1572.0, [156].log_data[7].valid := 1, [156].log_data[8].time := 1572.0, [156].log_data[8].valid := 1, [156].log_data[9].time := 1572.0, [156].log_data[9].valid := 1, [156].log_data[10].min := 1.0, [156].log_data[10].max := 1.0, [156].log_data[10].total := 1572.0, [156].log_data[10].time := 1572.0, [156].log_data[10].valid := 1, [156].log_data[11].time := 1572.0, [156].log_data[11].valid := 1, [156].log_data[12].min := 1.0, [156].log_data[12].max := 1.0, [156].log_data[12].total := 1572.0, [156].log_data[12].time := 1572.0, [156].log_data[12].valid := 1, [156].log_data[13].min := 1.0, [156].log_data[13].max := 1.0, [156].log_data[13].total := 1572.0, [156].log_data[13].time := 1572.0, [156].log_data[13].valid := 1, [156].log_data[14].time := 1572.0, [156].log_data[14].valid := 1, [156].log_data[15].time := 1572.0, [156].log_data[15].valid := 1, [156].log_data[16].time := 1572.0, [156].log_data[16].valid := 1, [156].log_data[17].min := 1.0, [156].log_data[17].max := 1.0, [156].log_data[17].total := 1572.0, [156].log_data[17].time := 1572.0, [156].log_data[17].valid := 1, [156].log_data[18].max := 1.0, [156].log_data[18].total := 487.00198, [156].log_data[18].time := 1572.0, [156].log_data[18].valid := 1, [156].log_data[19].max := 1.0, [156].log_data[19].total := 153.5, [156].log_data[19].time := 1572.0, [156].log_data[19].valid := 1, [156].log_data[20].time := 1572.0, [156].log_data[20].valid := 1, [156].log_data[21].min := 1.0, [156].log_data[21].max := 1.0, [156].log_data[21].total := 1572.0, [156].log_data[21].time := 1572.0, [156].log_data[21].valid := 1, [156].log_data[22].time := 1572.0, [156].log_data[22].valid := 1, [156].log_data[23].time := 1572.0, [156].log_data[23].valid := 1, [156].log_data[24].time := 1572.0, [156].log_data[24].valid := 1, [156].log_data[25].time := 1572.0, [156].log_data[25].valid := 1, [156].log_data[26].time := 1572.0,
        [156].log_data[26].valid := 1, [156].log_data[27].time := 1572.0, [156].log_data[27].valid := 1, [156].log_data[28].time := 1572.0, [156].log_data[28].valid := 1, [156].log_data[29].min := 1.0, [156].log_data[29].max := 1.0, [156].log_data[29].total := 1572.0, [156].log_data[29].time := 1572.0, [156].log_data[29].valid := 1, [156].log_data[30].min := 1.0, [156].log_data[30].max := 1.0, [156].log_data[30].total := 1572.0, [156].log_data[30].time := 1572.0, [156].log_data[30].valid := 1, [156].log_data[31].time := 1572.0, [156].log_data[31].valid := 1, [156].log_data[32].time := 1572.0, [156].log_data[32].valid := 1, [156].log_data[33].time := 1572.0, [156].log_data[33].valid := 1, [156].log_data[34].time := 1572.0, [156].log_data[34].valid := 1, [156].log_data[35].time := 1572.0, [156].log_data[35].valid := 1, [156].log_data[36].time := 1572.0, [156].log_data[36].valid := 1, [156].log_data[37].max := 7.285092, [156].log_data[37].total := 1016.4652, [156].log_data[37].time := 1572.0, [156].log_data[37].maxminute := 25, [156].log_data[37].valid := 1, [156].log_data[38].time := 1572.0, [156].log_data[38].valid := 1, [156].log_data[39].min := 0.9950596, [156].log_data[39].max := 1.0173191, [156].log_data[39].total := 1574.0399, [156].log_data[39].time := 1572.0, [156].log_data[39].minminute := 1, [156].log_data[39].maxminute := 26, [156].log_data[39].valid := 1, [156].log_data[40].min := 7.609111, [156].log_data[40].max := 7.6212025, [156].log_data[40].total := 11971.367, [156].log_data[40].time := 1572.0, [156].log_data[40].minminute := 23, [156].log_data[40].maxminute := 3, [156].log_data[40].valid := 1, [156].log_data[41].min := 0.021558594, [156].log_data[41].max := 0.022540038, [156].log_data[41].total := 34.5142, [156].log_data[41].time := 1572.0, [156].log_data[41].minminute := 6, [156].log_data[41].valid := 1, [156].log_data[42].min := 2.2908182, [156].log_data[42].max := 2.296118, [156].log_data[42].total := 3605.4492, [156].log_data[42].time := 1572.0, [156].log_data[42].minminute := 19, [156].log_data[42].maxminute := 19,
        [156].log_data[42].valid := 1, [156].log_data[43].min := -0.19999695, [156].log_data[43].max := -0.19999695, [156].log_data[43].total := -314.40942, [156].log_data[43].time := 1572.0, [156].log_data[43].valid := 1, [156].log_data[44].min := -0.27999878, [156].log_data[44].max := -0.22000122, [156].log_data[44].total := -351.34607, [156].log_data[44].time := 1572.0, [156].log_data[44].valid := 1, [156].log_data[45].time := 1572.0, [156].log_data[45].valid := 1, [156].log_data[46].time := 1572.0, [156].log_data[46].valid := 1, [156].log_data[47].time := 1572.0, [156].log_data[47].valid := 1, [156].log_data[48].min := 6.7385187, [156].log_data[48].max := 6.7489614, [156].log_data[48].total := 10601.376, [156].log_data[48].time := 1572.0, [156].log_data[48].maxminute := 25, [156].log_data[48].valid := 1, [156].log_data[49].min := 9.476719, [156].log_data[49].max := 9.5238285, [156].log_data[49].total := 14929.202, [156].log_data[49].time := 1572.0, [156].log_data[49].minminute := 11, [156].log_data[49].maxminute := 20, [156].log_data[49].valid := 1, [156].log_data[50].min := 2.0968432, [156].log_data[50].max := 2.1081495, [156].log_data[50].total := 3306.7727, [156].log_data[50].time := 1572.0, [156].log_data[50].maxminute := 24, [156].log_data[50].valid := 1, [156].log_data[51].time := 1572.0, [156].log_data[51].valid := 1, [156].log_data[52].min := -1.4800034, [156].log_data[52].max := -1.3600006, [156].log_data[52].total := -2244.1072, [156].log_data[52].time := 1572.0, [156].log_data[52].minminute := 23, [156].log_data[52].valid := 1, [156].log_data[53].min := -1.4400024, [156].log_data[53].max := -1.3199997, [156].log_data[53].total := -2173.8213, [156].log_data[53].time := 1572.0, [156].log_data[53].minminute := 7, [156].log_data[53].maxminute := 1, [156].log_data[53].valid := 1, [156].log_data[54].time := 1572.0, [156].log_data[54].valid := 1, [156].log_data[55].time := 1572.0, [156].log_data[55].valid := 1, [156].log_data[56].min := 0.15891084, [156].log_data[56].max := 0.15926416, [156].log_data[56].total := 250.03407, [156].log_data[56].time := 1572.0, [156].log_data[56].minminute := 2,
        [156].log_data[56].valid := 1, [156].log_data[57].min := 0.18619531, [156].log_data[57].max := 0.18658794, [156].log_data[57].total := 292.95258, [156].log_data[57].time := 1572.0, [156].log_data[57].minminute := 4, [156].log_data[57].maxminute := 14, [156].log_data[57].valid := 1, [156].log_data[58].time := 1572.0, [156].log_data[58].valid := 1, [156].log_data[59].time := 1572.0, [156].log_data[59].valid := 1, [156].log_data[60].time := 1572.0, [156].log_data[60].valid := 1, [156].log_data[61].valid := 1, [156].log_data[62].valid := 1, [156].log_data[63].valid := 1, [156].log_data[64].valid := 1, [156].log_data[65].valid := 1, [156].log_data[66].valid := 1, [156].log_data[67].valid := 1, [156].log_data[68].valid := 1, [156].log_data[69].valid := 1, [156].log_data[70].valid := 1, [156].log_data[71].valid := 1, [156].log_data[72].valid := 1, [156].log_data[73].valid := 1, [156].log_data[74].valid := 1, [156].log_data[75].valid := 1, [156].log_data[76].valid := 1, [156].log_data[77].valid := 1, [156].log_data[78].valid := 1, [156].log_data[79].valid := 1, [156].log_data[80].valid := 1, [156].log_data[81].valid := 1, [156].log_data[82].valid := 1, [156].log_data[83].valid := 1, [156].log_data[84].valid := 1, [156].log_data[85].valid := 1, [156].log_data[86].valid := 1, [156].log_data[87].valid := 1, [156].log_data[88].valid := 1, [156].log_data[89].valid := 1, [156].log_data[90].valid := 1, [156].log_data[91].valid := 1, [156].log_data[92].valid := 1, [156].log_data[93].valid := 1, [156].log_data[94].valid := 1, [156].log_data[95].valid := 1, [156].log_data[96].valid := 1, [156].log_data[97].valid := 1, [156].log_data[98].valid := 1, [156].log_data[99].valid := 1, [156].log_data[100].valid := 1, [156].log_data[101].valid := 1, [156].log_data[102].valid := 1, [156].log_data[103].valid := 1, [156].log_data[104].valid := 1, [156].log_data[105].valid := 1, [156].log_data[106].valid := 1,
        [156].log_data[107].valid := 1, [156].log_data[108].valid := 1, [156].log_data[109].valid := 1, [156].log_data[110].valid := 1, [156].log_data[111].valid := 1, [156].log_data[112].valid := 1, [156].log_data[113].valid := 1, [156].log_data[114].valid := 1, [156].log_data[115].valid := 1, [156].log_data[116].valid := 1, [156].log_data[117].valid := 1, [156].log_data[118].valid := 1, [156].log_data[119].valid := 1, [156].log_data[120].valid := 1, [156].log_data[121].valid := 1, [156].log_data[122].valid := 1, [156].log_data[123].valid := 1, [156].log_data[124].valid := 1, [157].log_data[0].min := 1.0, [157].log_data[0].max := 1.0, [157].log_data[0].total := 3600.0, [157].log_data[0].time := 3600.0, [157].log_data[0].valid := 1, [157].log_data[1].max := 1.0, [157].log_data[1].total := 122.249, [157].log_data[1].time := 3600.0, [157].log_data[1].maxminute := 57, [157].log_data[1].valid := 1, [157].log_data[2].max := 1.0, [157].log_data[2].total := 118.749, [157].log_data[2].time := 3600.0, [157].log_data[2].maxminute := 58, [157].log_data[2].valid := 1, [157].log_data[3].time := 3600.0, [157].log_data[3].valid := 1, [157].log_data[4].time := 3600.0, [157].log_data[4].valid := 1, [157].log_data[5].time := 3600.0, [157].log_data[5].valid := 1, [157].log_data[6].time := 3600.0, [157].log_data[6].valid := 1, [157].log_data[7].time := 3600.0, [157].log_data[7].valid := 1, [157].log_data[8].min := 1.0, [157].log_data[8].max := 1.0, [157].log_data[8].total := 3600.0, [157].log_data[8].time := 3600.0, [157].log_data[8].valid := 1, [157].log_data[9].min := 1.0, [157].log_data[9].max := 1.0, [157].log_data[9].total := 3600.0, [157].log_data[9].time := 3600.0, [157].log_data[9].valid := 1, [157].log_data[10].min := 1.0, [157].log_data[10].max := 1.0, [157].log_data[10].total := 3600.0, [157].log_data[10].time := 3600.0, [157].log_data[10].valid := 1, [157].log_data[11].time := 3600.0, [157].log_data[11].valid := 1,
        [157].log_data[12].min := 1.0, [157].log_data[12].max := 1.0, [157].log_data[12].total := 3600.0, [157].log_data[12].time := 3600.0, [157].log_data[12].valid := 1, [157].log_data[13].min := 1.0, [157].log_data[13].max := 1.0, [157].log_data[13].total := 3600.0, [157].log_data[13].time := 3600.0, [157].log_data[13].valid := 1, [157].log_data[14].time := 3600.0, [157].log_data[14].valid := 1, [157].log_data[15].time := 3600.0, [157].log_data[15].valid := 1, [157].log_data[16].time := 3600.0, [157].log_data[16].valid := 1, [157].log_data[17].min := 1.0, [157].log_data[17].max := 1.0, [157].log_data[17].total := 3600.0, [157].log_data[17].time := 3600.0, [157].log_data[17].valid := 1, [157].log_data[18].time := 3600.0, [157].log_data[18].valid := 1, [157].log_data[19].time := 3600.0, [157].log_data[19].valid := 1, [157].log_data[20].time := 3600.0, [157].log_data[20].valid := 1, [157].log_data[21].min := 1.0, [157].log_data[21].max := 1.0, [157].log_data[21].total := 3600.0, [157].log_data[21].time := 3600.0, [157].log_data[21].valid := 1, [157].log_data[22].time := 3600.0, [157].log_data[22].valid := 1, [157].log_data[23].time := 3600.0, [157].log_data[23].valid := 1, [157].log_data[24].time := 3600.0, [157].log_data[24].valid := 1, [157].log_data[25].time := 3600.0, [157].log_data[25].valid := 1, [157].log_data[26].time := 3600.0, [157].log_data[26].valid := 1, [157].log_data[27].time := 3600.0, [157].log_data[27].valid := 1, [157].log_data[28].time := 3600.0, [157].log_data[28].valid := 1, [157].log_data[29].min := 1.0, [157].log_data[29].max := 1.0, [157].log_data[29].total := 3600.0, [157].log_data[29].time := 3600.0, [157].log_data[29].valid := 1, [157].log_data[30].min := 1.0, [157].log_data[30].max := 1.0, [157].log_data[30].total := 3600.0, [157].log_data[30].time := 3600.0, [157].log_data[30].valid := 1, [157].log_data[31].max := 1.0, [157].log_data[31].total := 1629.998, [157].log_data[31].time := 3600.0, [157].log_data[31].maxminute := 1,
        [157].log_data[31].valid := 1, [157].log_data[32].max := 1.0, [157].log_data[32].total := 1440.7471, [157].log_data[32].time := 3600.0, [157].log_data[32].valid := 1, [157].log_data[33].time := 3600.0, [157].log_data[33].valid := 1, [157].log_data[34].time := 3600.0, [157].log_data[34].valid := 1, [157].log_data[35].max := 1.0, [157].log_data[35].total := 1629.7471, [157].log_data[35].time := 3600.0, [157].log_data[35].maxminute := 3, [157].log_data[35].valid := 1, [157].log_data[36].max := 1.0, [157].log_data[36].total := 1440.7471, [157].log_data[36].time := 3600.0, [157].log_data[36].minminute := 2, [157].log_data[36].valid := 1, [157].log_data[37].max := 7.633705, [157].log_data[37].total := 908.7482, [157].log_data[37].time := 3600.0, [157].log_data[37].maxminute := 59, [157].log_data[37].valid := 1, [157].log_data[38].time := 3600.0, [157].log_data[38].valid := 1, [157].log_data[39].min := 0.9941174, [157].log_data[39].max := 1.0143745, [157].log_data[39].total := 3598.8125, [157].log_data[39].time := 3600.0, [157].log_data[39].minminute := 32, [157].log_data[39].maxminute := 59, [157].log_data[39].valid := 1, [157].log_data[40].min := 7.539859, [157].log_data[40].max := 7.5821795, [157].log_data[40].total := 27230.074, [157].log_data[40].time := 3600.0, [157].log_data[40].minminute := 43, [157].log_data[40].maxminute := 39, [157].log_data[40].valid := 1, [157].log_data[41].min := 0.09497167, [157].log_data[41].max := 0.1463999, [157].log_data[41].total := 405.10977, [157].log_data[41].time := 3600.0, [157].log_data[41].minminute := 28, [157].log_data[41].maxminute := 50, [157].log_data[41].valid := 1, [157].log_data[42].min := 2.2929382, [157].log_data[42].max := 2.2980025, [157].log_data[42].total := 8264.619, [157].log_data[42].time := 3600.0, [157].log_data[42].minminute := 15, [157].log_data[42].maxminute := 12, [157].log_data[42].valid := 1, [157].log_data[43].min := -0.26000214, [157].log_data[43].max := -0.26000214, [157].log_data[43].total := -935.9732, [157].log_data[43].time := 3600.0, [157].log_data[43].valid := 1, [157].log_data[44].min := -0.30000305,
        [157].log_data[44].max := -0.27999878, [157].log_data[44].total := -1011.3994, [157].log_data[44].time := 3600.0, [157].log_data[44].valid := 1, [157].log_data[45].time := 3600.0, [157].log_data[45].valid := 1, [157].log_data[46].time := 3600.0, [157].log_data[46].valid := 1, [157].log_data[47].time := 3600.0, [157].log_data[47].valid := 1, [157].log_data[48].min := 6.5766573, [157].log_data[48].max := 6.795404, [157].log_data[48].total := 24170.107, [157].log_data[48].time := 3600.0, [157].log_data[48].minminute := 13, [157].log_data[48].maxminute := 28, [157].log_data[48].valid := 1, [157].log_data[49].min := 6.880372, [157].log_data[49].max := 9.499291, [157].log_data[49].total := 30221.293, [157].log_data[49].time := 3600.0, [157].log_data[49].minminute := 11, [157].log_data[49].maxminute := 55, [157].log_data[49].valid := 1, [157].log_data[50].min := 2.0193472, [157].log_data[50].max := 2.1066184, [157].log_data[50].total := 7433.0244, [157].log_data[50].time := 3600.0, [157].log_data[50].minminute := 59, [157].log_data[50].maxminute := 1, [157].log_data[50].valid := 1, [157].log_data[51].time := 3600.0, [157].log_data[51].valid := 1, [157].log_data[52].min := -2.7799988, [157].log_data[52].max := 0.13999939, [157].log_data[52].total := -7446.465, [157].log_data[52].time := 3600.0, [157].log_data[52].minminute := 12, [157].log_data[52].maxminute := 32, [157].log_data[52].valid := 1, [157].log_data[53].min := -2.2400055, [157].log_data[53].max := 0.8800049, [157].log_data[53].total := -5907.595, [157].log_data[53].time := 3600.0, [157].log_data[53].minminute := 25, [157].log_data[53].maxminute := 3, [157].log_data[53].valid := 1, [157].log_data[54].max := 0.53, [157].log_data[54].total := 1217.3512, [157].log_data[54].time := 3600.0, [157].log_data[54].maxminute := 22, [157].log_data[54].valid := 1, [157].log_data[55].max := 0.537, [157].log_data[55].total := 1217.0703, [157].log_data[55].time := 3600.0, [157].log_data[55].minminute := 2, [157].log_data[55].maxminute := 3, [157].log_data[55].valid := 1, [157].log_data[56].min := 0.16079521, [157].log_data[56].max := 0.16122705,
        [157].log_data[56].total := 579.4577, [157].log_data[56].time := 3600.0, [157].log_data[56].minminute := 6, [157].log_data[56].maxminute := 48, [157].log_data[56].valid := 1, [157].log_data[57].min := 0.3606984, [157].log_data[57].max := 0.36262202, [157].log_data[57].total := 1300.5449, [157].log_data[57].time := 3600.0, [157].log_data[57].minminute := 24, [157].log_data[57].maxminute := 2, [157].log_data[57].valid := 1, [157].log_data[58].time := 3600.0, [157].log_data[58].valid := 1, [157].log_data[59].time := 3600.0, [157].log_data[59].valid := 1, [157].log_data[60].valid := 1, [157].log_data[61].valid := 1, [157].log_data[62].valid := 1, [157].log_data[63].valid := 1, [157].log_data[64].valid := 1, [157].log_data[65].valid := 1, [157].log_data[66].valid := 1, [157].log_data[67].valid := 1, [157].log_data[68].valid := 1, [157].log_data[69].valid := 1, [157].log_data[70].valid := 1, [157].log_data[71].valid := 1, [157].log_data[72].valid := 1, [157].log_data[73].valid := 1, [157].log_data[74].valid := 1, [157].log_data[75].valid := 1, [157].log_data[76].valid := 1, [157].log_data[77].valid := 1, [157].log_data[78].valid := 1, [157].log_data[79].valid := 1, [157].log_data[80].valid := 1, [157].log_data[81].valid := 1, [157].log_data[82].valid := 1, [157].log_data[83].valid := 1, [157].log_data[84].valid := 1, [157].log_data[85].valid := 1, [157].log_data[86].valid := 1, [157].log_data[87].valid := 1, [157].log_data[88].valid := 1, [157].log_data[89].valid := 1, [157].log_data[90].valid := 1, [157].log_data[91].valid := 1, [157].log_data[92].valid := 1, [157].log_data[93].valid := 1, [157].log_data[94].valid := 1, [157].log_data[95].valid := 1, [157].log_data[96].valid := 1, [157].log_data[97].valid := 1, [157].log_data[98].valid := 1, [157].log_data[99].valid := 1, [157].log_data[100].valid := 1, [157].log_data[101].valid := 1, [157].log_data[102].valid := 1, [157].log_data[103].valid := 1,
        [157].log_data[104].valid := 1, [157].log_data[105].valid := 1, [157].log_data[106].valid := 1, [157].log_data[107].valid := 1, [157].log_data[108].valid := 1, [157].log_data[109].valid := 1, [157].log_data[110].valid := 1, [157].log_data[111].valid := 1, [157].log_data[112].valid := 1, [157].log_data[113].valid := 1, [157].log_data[114].valid := 1, [157].log_data[115].valid := 1, [157].log_data[116].valid := 1, [157].log_data[117].valid := 1, [157].log_data[118].valid := 1, [157].log_data[119].valid := 1, [157].log_data[120].valid := 1, [157].log_data[121].valid := 1, [157].log_data[122].valid := 1, [157].log_data[123].valid := 1, [157].log_data[124].valid := 1, [157].time.Year := 2023, [157].time.Month := 1, [157].time.Day := 11, [157].time.Hour := 8, [157].time.Minute := 59, [157].time.Second := 59, [158].log_data[0].min := 1.0, [158].log_data[0].max := 1.0, [158].log_data[0].total := 3600.0, [158].log_data[0].time := 3600.0, [158].log_data[0].valid := 1, [158].log_data[1].max := 1.0, [158].log_data[1].total := 425.251, [158].log_data[1].time := 3600.0, [158].log_data[1].minminute := 7, [158].log_data[1].valid := 1, [158].log_data[2].max := 1.0, [158].log_data[2].total := 425.251, [158].log_data[2].time := 3600.0, [158].log_data[2].minminute := 7, [158].log_data[2].valid := 1, [158].log_data[3].time := 3600.0, [158].log_data[3].valid := 1, [158].log_data[4].time := 3600.0, [158].log_data[4].valid := 1, [158].log_data[5].max := 1.0, [158].log_data[5].total := 238.0, [158].log_data[5].time := 3600.0, [158].log_data[5].valid := 1, [158].log_data[6].time := 3600.0, [158].log_data[6].valid := 1, [158].log_data[7].time := 3600.0, [158].log_data[7].valid := 1, [158].log_data[8].min := 1.0, [158].log_data[8].max := 1.0, [158].log_data[8].total := 3600.0, [158].log_data[8].time := 3600.0, [158].log_data[8].valid := 1, [158].log_data[9].min := 1.0,
        [158].log_data[9].max := 1.0, [158].log_data[9].total := 3600.0, [158].log_data[9].time := 3600.0, [158].log_data[9].valid := 1, [158].log_data[10].min := 1.0, [158].log_data[10].max := 1.0, [158].log_data[10].total := 3600.0, [158].log_data[10].time := 3600.0, [158].log_data[10].valid := 1, [158].log_data[11].time := 3600.0, [158].log_data[11].valid := 1, [158].log_data[12].min := 1.0, [158].log_data[12].max := 1.0, [158].log_data[12].total := 3600.0, [158].log_data[12].time := 3600.0, [158].log_data[12].valid := 1, [158].log_data[13].min := 1.0, [158].log_data[13].max := 1.0, [158].log_data[13].total := 3600.0, [158].log_data[13].time := 3600.0, [158].log_data[13].valid := 1, [158].log_data[14].time := 3600.0, [158].log_data[14].valid := 1, [158].log_data[15].time := 3600.0, [158].log_data[15].valid := 1, [158].log_data[16].time := 3600.0, [158].log_data[16].valid := 1, [158].log_data[17].min := 1.0, [158].log_data[17].max := 1.0, [158].log_data[17].total := 3600.0, [158].log_data[17].time := 3600.0, [158].log_data[17].valid := 1, [158].log_data[18].time := 3600.0, [158].log_data[18].valid := 1, [158].log_data[19].time := 3600.0, [158].log_data[19].valid := 1, [158].log_data[20].time := 3600.0, [158].log_data[20].valid := 1, [158].log_data[21].min := 1.0, [158].log_data[21].max := 1.0, [158].log_data[21].total := 3600.0, [158].log_data[21].time := 3600.0, [158].log_data[21].valid := 1, [158].log_data[22].time := 3600.0, [158].log_data[22].valid := 1, [158].log_data[23].time := 3600.0, [158].log_data[23].valid := 1, [158].log_data[24].time := 3600.0, [158].log_data[24].valid := 1, [158].log_data[25].time := 3600.0, [158].log_data[25].valid := 1, [158].log_data[26].time := 3600.0, [158].log_data[26].valid := 1, [158].log_data[27].time := 3600.0, [158].log_data[27].valid := 1, [158].log_data[28].time := 3600.0, [158].log_data[28].valid := 1, [158].log_data[29].min := 1.0, [158].log_data[29].max := 1.0, [158].log_data[29].total := 3600.0,
        [158].log_data[29].time := 3600.0, [158].log_data[29].valid := 1, [158].log_data[30].min := 1.0, [158].log_data[30].max := 1.0, [158].log_data[30].total := 3600.0, [158].log_data[30].time := 3600.0, [158].log_data[30].valid := 1, [158].log_data[31].max := 1.0, [158].log_data[31].total := 1629.7471, [158].log_data[31].time := 3600.0, [158].log_data[31].maxminute := 4, [158].log_data[31].valid := 1, [158].log_data[32].max := 1.0, [158].log_data[32].total := 1440.998, [158].log_data[32].time := 3600.0, [158].log_data[32].minminute := 3, [158].log_data[32].valid := 1, [158].log_data[33].time := 3600.0, [158].log_data[33].valid := 1, [158].log_data[34].time := 3600.0, [158].log_data[34].valid := 1, [158].log_data[35].max := 1.0, [158].log_data[35].total := 1629.7471, [158].log_data[35].time := 3600.0, [158].log_data[35].maxminute := 6, [158].log_data[35].valid := 1, [158].log_data[36].max := 1.0, [158].log_data[36].total := 1440.7471, [158].log_data[36].time := 3600.0, [158].log_data[36].minminute := 5, [158].log_data[36].valid := 1, [158].log_data[37].max := 7.62978, [158].log_data[37].total := 2725.4233, [158].log_data[37].time := 3600.0, [158].log_data[37].minminute := 6, [158].log_data[37].valid := 1, [158].log_data[38].time := 3600.0, [158].log_data[38].valid := 1, [158].log_data[39].min := 0.9961195, [158].log_data[39].max := 1.0210879, [158].log_data[39].total := 3607.727, [158].log_data[39].time := 3600.0, [158].log_data[39].minminute := 15, [158].log_data[39].maxminute := 4, [158].log_data[39].valid := 1, [158].log_data[40].min := 7.5373855, [158].log_data[40].max := 7.5819044, [158].log_data[40].total := 27230.795, [158].log_data[40].time := 3600.0, [158].log_data[40].minminute := 55, [158].log_data[40].maxminute := 41, [158].log_data[40].valid := 1, [158].log_data[41].min := 0.11656372, [158].log_data[41].max := 0.14325929, [158].log_data[41].total := 470.01544, [158].log_data[41].time := 3600.0, [158].log_data[41].minminute := 53, [158].log_data[41].maxminute := 33, [158].log_data[41].valid := 1, [158].log_data[42].min := 2.2928205,
        [158].log_data[42].max := 2.298238, [158].log_data[42].total := 8264.55, [158].log_data[42].time := 3600.0, [158].log_data[42].minminute := 8, [158].log_data[42].maxminute := 30, [158].log_data[42].valid := 1, [158].log_data[43].min := -0.26000214, [158].log_data[43].max := -0.23999786, [158].log_data[43].total := -935.9682, [158].log_data[43].time := 3600.0, [158].log_data[43].maxminute := 51, [158].log_data[43].valid := 1, [158].log_data[44].min := -0.30000305, [158].log_data[44].max := -0.27999878, [158].log_data[44].total := -1007.94684, [158].log_data[44].time := 3600.0, [158].log_data[44].minminute := 10, [158].log_data[44].valid := 1, [158].log_data[45].time := 3600.0, [158].log_data[45].valid := 1, [158].log_data[46].time := 3600.0, [158].log_data[46].valid := 1, [158].log_data[47].time := 3600.0, [158].log_data[47].valid := 1, [158].log_data[48].min := 6.575283, [158].log_data[48].max := 6.9108233, [158].log_data[48].total := 24212.799, [158].log_data[48].time := 3600.0, [158].log_data[48].minminute := 27, [158].log_data[48].maxminute := 7, [158].log_data[48].valid := 1, [158].log_data[49].min := 6.9537854, [158].log_data[49].max := 9.494385, [158].log_data[49].total := 29306.541, [158].log_data[49].time := 3600.0, [158].log_data[49].minminute := 21, [158].log_data[49].valid := 1, [158].log_data[50].min := 2.0192294, [158].log_data[50].max := 2.1346488, [158].log_data[50].total := 7538.001, [158].log_data[50].time := 3600.0, [158].log_data[50].maxminute := 7, [158].log_data[50].valid := 1, [158].log_data[51].time := 3600.0, [158].log_data[51].valid := 1, [158].log_data[52].min := -2.800003, [158].log_data[52].max := 0.13999939, [158].log_data[52].total := -7479.4966, [158].log_data[52].time := 3600.0, [158].log_data[52].minminute := 25, [158].log_data[52].maxminute := 3, [158].log_data[52].valid := 1, [158].log_data[53].min := -2.380005, [158].log_data[53].max := 0.8200073, [158].log_data[53].total := -6003.276, [158].log_data[53].time := 3600.0, [158].log_data[53].minminute := 49, [158].log_data[53].maxminute := 6, [158].log_data[53].valid := 1, [158].log_data[54].max := 0.5075,
        [158].log_data[54].total := 1217.0332, [158].log_data[54].time := 3600.0, [158].log_data[54].minminute := 3, [158].log_data[54].maxminute := 36, [158].log_data[54].valid := 1, [158].log_data[55].max := 0.5545, [158].log_data[55].total := 1217.2241, [158].log_data[55].time := 3600.0, [158].log_data[55].minminute := 5, [158].log_data[55].maxminute := 49, [158].log_data[55].valid := 1, [158].log_data[56].min := 0.16079521, [158].log_data[56].max := 0.1611878, [158].log_data[56].total := 579.4338, [158].log_data[56].time := 3600.0, [158].log_data[56].minminute := 24, [158].log_data[56].maxminute := 5, [158].log_data[56].valid := 1, [158].log_data[57].min := 0.35912803, [158].log_data[57].max := 0.3610517, [158].log_data[57].total := 1296.2554, [158].log_data[57].time := 3600.0, [158].log_data[57].minminute := 56, [158].log_data[57].valid := 1, [158].log_data[58].time := 3600.0, [158].log_data[58].valid := 1, [158].log_data[59].time := 3600.0, [158].log_data[59].valid := 1, [158].log_data[60].valid := 1, [158].log_data[61].valid := 1, [158].log_data[62].valid := 1, [158].log_data[63].valid := 1, [158].log_data[64].valid := 1, [158].log_data[65].valid := 1, [158].log_data[66].valid := 1, [158].log_data[67].valid := 1, [158].log_data[68].valid := 1, [158].log_data[69].valid := 1, [158].log_data[70].valid := 1, [158].log_data[71].valid := 1, [158].log_data[72].valid := 1, [158].log_data[73].valid := 1, [158].log_data[74].valid := 1, [158].log_data[75].valid := 1, [158].log_data[76].valid := 1, [158].log_data[77].valid := 1, [158].log_data[78].valid := 1, [158].log_data[79].valid := 1, [158].log_data[80].valid := 1, [158].log_data[81].valid := 1, [158].log_data[82].valid := 1, [158].log_data[83].valid := 1, [158].log_data[84].valid := 1, [158].log_data[85].valid := 1, [158].log_data[86].valid := 1, [158].log_data[87].valid := 1, [158].log_data[88].valid := 1, [158].log_data[89].valid := 1, [158].log_data[90].valid := 1, [158].log_data[91].valid := 1,
        [158].log_data[92].valid := 1, [158].log_data[93].valid := 1, [158].log_data[94].valid := 1, [158].log_data[95].valid := 1, [158].log_data[96].valid := 1, [158].log_data[97].valid := 1, [158].log_data[98].valid := 1, [158].log_data[99].valid := 1, [158].log_data[100].valid := 1, [158].log_data[101].valid := 1, [158].log_data[102].valid := 1, [158].log_data[103].valid := 1, [158].log_data[104].valid := 1, [158].log_data[105].valid := 1, [158].log_data[106].valid := 1, [158].log_data[107].valid := 1, [158].log_data[108].valid := 1, [158].log_data[109].valid := 1, [158].log_data[110].valid := 1, [158].log_data[111].valid := 1, [158].log_data[112].valid := 1, [158].log_data[113].valid := 1, [158].log_data[114].valid := 1, [158].log_data[115].valid := 1, [158].log_data[116].valid := 1, [158].log_data[117].valid := 1, [158].log_data[118].valid := 1, [158].log_data[119].valid := 1, [158].log_data[120].valid := 1, [158].log_data[121].valid := 1, [158].log_data[122].valid := 1, [158].log_data[123].valid := 1, [158].log_data[124].valid := 1, [158].time.Year := 2023, [158].time.Month := 1, [158].time.Day := 11, [158].time.Hour := 9, [158].time.Minute := 59, [158].time.Second := 59, [159].log_data[0].min := 1.0, [159].log_data[0].max := 1.0, [159].log_data[0].total := 3600.0, [159].log_data[0].time := 3600.0, [159].log_data[0].valid := 1, [159].log_data[1].max := 1.0, [159].log_data[1].total := 766.0, [159].log_data[1].time := 3600.0, [159].log_data[1].maxminute := 22, [159].log_data[1].valid := 1, [159].log_data[2].max := 1.0, [159].log_data[2].total := 759.0, [159].log_data[2].time := 3600.0, [159].log_data[2].maxminute := 22, [159].log_data[2].valid := 1, [159].log_data[3].time := 3600.0, [159].log_data[3].valid := 1, [159].log_data[4].time := 3600.0, [159].log_data[4].valid := 1, [159].log_data[5].max := 1.0, [159].log_data[5].total := 240.5,
        [159].log_data[5].time := 3600.0, [159].log_data[5].maxminute := 25, [159].log_data[5].valid := 1, [159].log_data[6].time := 3600.0, [159].log_data[6].valid := 1, [159].log_data[7].time := 3600.0, [159].log_data[7].valid := 1, [159].log_data[8].max := 1.0, [159].log_data[8].total := 3572.749, [159].log_data[8].time := 3600.0, [159].log_data[8].minminute := 5, [159].log_data[8].valid := 1, [159].log_data[9].max := 1.0, [159].log_data[9].total := 3569.249, [159].log_data[9].time := 3600.0, [159].log_data[9].minminute := 5, [159].log_data[9].valid := 1, [159].log_data[10].min := 1.0, [159].log_data[10].max := 1.0, [159].log_data[10].total := 3600.0, [159].log_data[10].time := 3600.0, [159].log_data[10].valid := 1, [159].log_data[11].time := 3600.0, [159].log_data[11].valid := 1, [159].log_data[12].min := 1.0, [159].log_data[12].max := 1.0, [159].log_data[12].total := 3600.0, [159].log_data[12].time := 3600.0, [159].log_data[12].valid := 1, [159].log_data[13].min := 1.0, [159].log_data[13].max := 1.0, [159].log_data[13].total := 3600.0, [159].log_data[13].time := 3600.0, [159].log_data[13].valid := 1, [159].log_data[14].time := 3600.0, [159].log_data[14].valid := 1, [159].log_data[15].time := 3600.0, [159].log_data[15].valid := 1, [159].log_data[16].time := 3600.0, [159].log_data[16].valid := 1, [159].log_data[17].max := 1.0, [159].log_data[17].total := 3565.5, [159].log_data[17].time := 3600.0, [159].log_data[17].minminute := 5, [159].log_data[17].valid := 1, [159].log_data[18].time := 3600.0, [159].log_data[18].valid := 1, [159].log_data[19].time := 3600.0, [159].log_data[19].valid := 1, [159].log_data[20].time := 3600.0, [159].log_data[20].valid := 1, [159].log_data[21].max := 1.0, [159].log_data[21].total := 3562.249, [159].log_data[21].time := 3600.0, [159].log_data[21].minminute := 5, [159].log_data[21].valid := 1, [159].log_data[22].time := 3600.0, [159].log_data[22].valid := 1, [159].log_data[23].time := 3600.0, [159].log_data[23].valid := 1,
        [159].log_data[24].time := 3600.0, [159].log_data[24].valid := 1, [159].log_data[25].time := 3600.0, [159].log_data[25].valid := 1, [159].log_data[26].time := 3600.0, [159].log_data[26].valid := 1, [159].log_data[27].time := 3600.0, [159].log_data[27].valid := 1, [159].log_data[28].time := 3600.0, [159].log_data[28].valid := 1, [159].log_data[29].max := 1.0, [159].log_data[29].total := 3558.749, [159].log_data[29].time := 3600.0, [159].log_data[29].minminute := 5, [159].log_data[29].valid := 1, [159].log_data[30].max := 1.0, [159].log_data[30].total := 3555.249, [159].log_data[30].time := 3600.0, [159].log_data[30].minminute := 5, [159].log_data[30].valid := 1, [159].log_data[31].max := 1.0, [159].log_data[31].total := 1383.0, [159].log_data[31].time := 3600.0, [159].log_data[31].maxminute := 12, [159].log_data[31].valid := 1, [159].log_data[32].max := 1.0, [159].log_data[32].total := 1466.749, [159].log_data[32].time := 3600.0, [159].log_data[32].minminute := 5, [159].log_data[32].valid := 1, [159].log_data[33].time := 3600.0, [159].log_data[33].valid := 1, [159].log_data[34].time := 3600.0, [159].log_data[34].valid := 1, [159].log_data[35].max := 1.0, [159].log_data[35].total := 1248.2471, [159].log_data[35].time := 3600.0, [159].log_data[35].maxminute := 15, [159].log_data[35].valid := 1, [159].log_data[36].max := 1.0, [159].log_data[36].total := 1598.749, [159].log_data[36].time := 3600.0, [159].log_data[36].minminute := 5, [159].log_data[36].valid := 1, [159].log_data[37].max := 7.396193, [159].log_data[37].total := 4492.3228, [159].log_data[37].time := 3600.0, [159].log_data[37].maxminute := 38, [159].log_data[37].valid := 1, [159].log_data[38].time := 3600.0, [159].log_data[38].valid := 1, [159].log_data[39].min := 0.9950596, [159].log_data[39].max := 1.0212055, [159].log_data[39].total := 3627.762, [159].log_data[39].time := 3600.0, [159].log_data[39].minminute := 32, [159].log_data[39].maxminute := 25, [159].log_data[39].valid := 1, [159].log_data[40].min := 7.5459046, [159].log_data[40].max := 7.5777817,
        [159].log_data[40].total := 27246.963, [159].log_data[40].time := 3600.0, [159].log_data[40].minminute := 3, [159].log_data[40].maxminute := 11, [159].log_data[40].valid := 1, [159].log_data[41].min := 0.11970434, [159].log_data[41].max := 0.13128565, [159].log_data[41].total := 450.94684, [159].log_data[41].time := 3600.0, [159].log_data[41].minminute := 59, [159].log_data[41].maxminute := 23, [159].log_data[41].valid := 1, [159].log_data[42].min := 2.292467, [159].log_data[42].max := 2.2987092, [159].log_data[42].total := 8264.462, [159].log_data[42].time := 3600.0, [159].log_data[42].minminute := 9, [159].log_data[42].maxminute := 37, [159].log_data[42].valid := 1, [159].log_data[43].min := -0.26000214, [159].log_data[43].max := -0.23999786, [159].log_data[43].total := -880.5832, [159].log_data[43].time := 3600.0, [159].log_data[43].maxminute := 9, [159].log_data[43].valid := 1, [159].log_data[44].min := -0.30000305, [159].log_data[44].max := -0.26000214, [159].log_data[44].total := -969.44635, [159].log_data[44].time := 3600.0, [159].log_data[44].minminute := 5, [159].log_data[44].maxminute := 15, [159].log_data[44].valid := 1, [159].log_data[45].time := 3600.0, [159].log_data[45].valid := 1, [159].log_data[46].time := 3600.0, [159].log_data[46].valid := 1, [159].log_data[47].time := 3600.0, [159].log_data[47].valid := 1, [159].log_data[48].min := 6.5766573, [159].log_data[48].max := 6.9476476, [159].log_data[48].total := 24196.08, [159].log_data[48].time := 3600.0, [159].log_data[48].minminute := 53, [159].log_data[48].maxminute := 27, [159].log_data[48].valid := 1, [159].log_data[49].min := 6.799893, [159].log_data[49].max := 9.521865, [159].log_data[49].total := 30186.838, [159].log_data[49].time := 3600.0, [159].log_data[49].minminute := 50, [159].log_data[49].maxminute := 24, [159].log_data[49].valid := 1, [159].log_data[50].min := 2.0233517, [159].log_data[50].max := 2.1421862, [159].log_data[50].total := 7513.9883, [159].log_data[50].time := 3600.0, [159].log_data[50].minminute := 23, [159].log_data[50].maxminute := 33, [159].log_data[50].valid := 1, [159].log_data[51].time := 3600.0,
        [159].log_data[51].valid := 1, [159].log_data[52].min := -2.8199997, [159].log_data[52].max := 0.13999939, [159].log_data[52].total := -6949.826, [159].log_data[52].time := 3600.0, [159].log_data[52].minminute := 13, [159].log_data[52].maxminute := 6, [159].log_data[52].valid := 1, [159].log_data[53].min := -2.6600037, [159].log_data[53].max := 0.2400055, [159].log_data[53].total := -6409.842, [159].log_data[53].time := 3600.0, [159].log_data[53].minminute := 57, [159].log_data[53].maxminute := 10, [159].log_data[53].valid := 1, [159].log_data[54].max := 0.513, [159].log_data[54].total := 1129.3976, [159].log_data[54].time := 3600.0, [159].log_data[54].minminute := 5, [159].log_data[54].maxminute := 44, [159].log_data[54].valid := 1, [159].log_data[55].max := 0.536, [159].log_data[55].total := 1128.0266, [159].log_data[55].time := 3600.0, [159].log_data[55].minminute := 5, [159].log_data[55].maxminute := 36, [159].log_data[55].valid := 1, [159].log_data[56].min := 0.16079521, [159].log_data[56].max := 0.16122705, [159].log_data[56].total := 579.5096, [159].log_data[56].time := 3600.0, [159].log_data[56].minminute := 6, [159].log_data[56].maxminute := 5, [159].log_data[56].valid := 1, [159].log_data[57].min := 0.3576755, [159].log_data[57].max := 0.3596384, [159].log_data[57].total := 1293.1948, [159].log_data[57].time := 3600.0, [159].log_data[57].minminute := 59, [159].log_data[57].maxminute := 48, [159].log_data[57].valid := 1, [159].log_data[58].time := 3600.0, [159].log_data[58].valid := 1, [159].log_data[59].time := 3600.0, [159].log_data[59].valid := 1, [159].log_data[60].valid := 1, [159].log_data[61].valid := 1, [159].log_data[62].valid := 1, [159].log_data[63].valid := 1, [159].log_data[64].valid := 1, [159].log_data[65].valid := 1, [159].log_data[66].valid := 1, [159].log_data[67].valid := 1, [159].log_data[68].valid := 1, [159].log_data[69].valid := 1, [159].log_data[70].valid := 1, [159].log_data[71].valid := 1, [159].log_data[72].valid := 1, [159].log_data[73].valid := 1, [159].log_data[74].valid := 1,
        [159].log_data[75].valid := 1, [159].log_data[76].valid := 1, [159].log_data[77].valid := 1, [159].log_data[78].valid := 1, [159].log_data[79].valid := 1, [159].log_data[80].valid := 1, [159].log_data[81].valid := 1, [159].log_data[82].valid := 1, [159].log_data[83].valid := 1, [159].log_data[84].valid := 1, [159].log_data[85].valid := 1, [159].log_data[86].valid := 1, [159].log_data[87].valid := 1, [159].log_data[88].valid := 1, [159].log_data[89].valid := 1, [159].log_data[90].valid := 1, [159].log_data[91].valid := 1, [159].log_data[92].valid := 1, [159].log_data[93].valid := 1, [159].log_data[94].valid := 1, [159].log_data[95].valid := 1, [159].log_data[96].valid := 1, [159].log_data[97].valid := 1, [159].log_data[98].valid := 1, [159].log_data[99].valid := 1, [159].log_data[100].valid := 1, [159].log_data[101].valid := 1, [159].log_data[102].valid := 1, [159].log_data[103].valid := 1, [159].log_data[104].valid := 1, [159].log_data[105].valid := 1, [159].log_data[106].valid := 1, [159].log_data[107].valid := 1, [159].log_data[108].valid := 1, [159].log_data[109].valid := 1, [159].log_data[110].valid := 1, [159].log_data[111].valid := 1, [159].log_data[112].valid := 1, [159].log_data[113].valid := 1, [159].log_data[114].valid := 1, [159].log_data[115].valid := 1, [159].log_data[116].valid := 1, [159].log_data[117].valid := 1, [159].log_data[118].valid := 1, [159].log_data[119].valid := 1, [159].log_data[120].valid := 1, [159].log_data[121].valid := 1, [159].log_data[122].valid := 1, [159].log_data[123].valid := 1, [159].log_data[124].valid := 1, [159].time.Year := 2023, [159].time.Month := 1, [159].time.Day := 11, [159].time.Hour := 10, [159].time.Minute := 59, [159].time.Second := 59, [160].log_data[0].min := 1.0, [160].log_data[0].max := 1.0, [160].log_data[0].total := 3600.0, [160].log_data[0].time := 3600.0,
        [160].log_data[0].valid := 1, [160].log_data[1].time := 3600.0, [160].log_data[1].valid := 1, [160].log_data[2].time := 3600.0, [160].log_data[2].valid := 1, [160].log_data[3].time := 3600.0, [160].log_data[3].valid := 1, [160].log_data[4].time := 3600.0, [160].log_data[4].valid := 1, [160].log_data[5].max := 1.0, [160].log_data[5].total := 61.5, [160].log_data[5].time := 3600.0, [160].log_data[5].maxminute := 42, [160].log_data[5].valid := 1, [160].log_data[6].time := 3600.0, [160].log_data[6].valid := 1, [160].log_data[7].time := 3600.0, [160].log_data[7].valid := 1, [160].log_data[8].max := 1.0, [160].log_data[8].total := 1848.0, [160].log_data[8].time := 3600.0, [160].log_data[8].minminute := 2, [160].log_data[8].valid := 1, [160].log_data[9].max := 1.0, [160].log_data[9].total := 1844.5, [160].log_data[9].time := 3600.0, [160].log_data[9].minminute := 2, [160].log_data[9].valid := 1, [160].log_data[10].min := 1.0, [160].log_data[10].max := 1.0, [160].log_data[10].total := 3600.0, [160].log_data[10].time := 3600.0, [160].log_data[10].valid := 1, [160].log_data[11].time := 3600.0, [160].log_data[11].valid := 1, [160].log_data[12].min := 1.0, [160].log_data[12].max := 1.0, [160].log_data[12].total := 3600.0, [160].log_data[12].time := 3600.0, [160].log_data[12].valid := 1, [160].log_data[13].min := 1.0, [160].log_data[13].max := 1.0, [160].log_data[13].total := 3600.0, [160].log_data[13].time := 3600.0, [160].log_data[13].valid := 1, [160].log_data[14].time := 3600.0, [160].log_data[14].valid := 1, [160].log_data[15].time := 3600.0, [160].log_data[15].valid := 1, [160].log_data[16].time := 3600.0, [160].log_data[16].valid := 1, [160].log_data[17].max := 1.0, [160].log_data[17].total := 3566.0, [160].log_data[17].time := 3600.0, [160].log_data[17].minminute := 2, [160].log_data[17].valid := 1, [160].log_data[18].time := 3600.0, [160].log_data[18].valid := 1, [160].log_data[19].time := 3600.0, [160].log_data[19].valid := 1,
        [160].log_data[20].time := 3600.0, [160].log_data[20].valid := 1, [160].log_data[21].max := 1.0, [160].log_data[21].total := 3562.5, [160].log_data[21].time := 3600.0, [160].log_data[21].minminute := 2, [160].log_data[21].valid := 1, [160].log_data[22].time := 3600.0, [160].log_data[22].valid := 1, [160].log_data[23].time := 3600.0, [160].log_data[23].valid := 1, [160].log_data[24].time := 3600.0, [160].log_data[24].valid := 1, [160].log_data[25].time := 3600.0, [160].log_data[25].valid := 1, [160].log_data[26].time := 3600.0, [160].log_data[26].valid := 1, [160].log_data[27].time := 3600.0, [160].log_data[27].valid := 1, [160].log_data[28].time := 3600.0, [160].log_data[28].valid := 1, [160].log_data[29].max := 1.0, [160].log_data[29].total := 3558.749, [160].log_data[29].time := 3600.0, [160].log_data[29].minminute := 2, [160].log_data[29].valid := 1, [160].log_data[30].max := 1.0, [160].log_data[30].total := 3555.249, [160].log_data[30].time := 3600.0, [160].log_data[30].minminute := 2, [160].log_data[30].valid := 1, [160].log_data[31].max := 1.0, [160].log_data[31].total := 789.498, [160].log_data[31].time := 3600.0, [160].log_data[31].minminute := 2, [160].log_data[31].valid := 1, [160].log_data[32].max := 1.0, [160].log_data[32].total := 543.5, [160].log_data[32].time := 3600.0, [160].log_data[32].maxminute := 10, [160].log_data[32].valid := 1, [160].log_data[33].max := 1.0, [160].log_data[33].total := 636.0, [160].log_data[33].time := 3600.0, [160].log_data[33].maxminute := 8, [160].log_data[33].valid := 1, [160].log_data[34].max := 1.0, [160].log_data[34].total := 643.749, [160].log_data[34].time := 3600.0, [160].log_data[34].maxminute := 8, [160].log_data[34].valid := 1, [160].log_data[35].max := 1.0, [160].log_data[35].total := 848.249, [160].log_data[35].time := 3600.0, [160].log_data[35].minminute := 2, [160].log_data[35].valid := 1, [160].log_data[36].max := 1.0, [160].log_data[36].total := 543.249, [160].log_data[36].time := 3600.0, [160].log_data[36].maxminute := 13,
        [160].log_data[36].valid := 1, [160].log_data[37].time := 3600.0, [160].log_data[37].valid := 1, [160].log_data[38].time := 3600.0, [160].log_data[38].valid := 1, [160].log_data[39].min := 0.9957663, [160].log_data[39].max := 1.0201455, [160].log_data[39].total := 3644.4578, [160].log_data[39].time := 3600.0, [160].log_data[39].minminute := 54, [160].log_data[39].maxminute := 2, [160].log_data[39].valid := 1, [160].log_data[40].min := 7.553049, [160].log_data[40].max := 7.5791564, [160].log_data[40].total := 27246.312, [160].log_data[40].time := 3600.0, [160].log_data[40].minminute := 54, [160].log_data[40].maxminute := 57, [160].log_data[40].valid := 1, [160].log_data[41].min := 0.089868166, [160].log_data[41].max := 0.14011866, [160].log_data[41].total := 423.66803, [160].log_data[41].time := 3600.0, [160].log_data[41].minminute := 51, [160].log_data[41].maxminute := 26, [160].log_data[41].valid := 1, [160].log_data[42].min := 2.2928205, [160].log_data[42].max := 2.2980025, [160].log_data[42].total := 8264.274, [160].log_data[42].time := 3600.0, [160].log_data[42].maxminute := 36, [160].log_data[42].valid := 1, [160].log_data[43].min := -0.26000214, [160].log_data[43].max := -0.22000122, [160].log_data[43].total := -863.711, [160].log_data[43].time := 3600.0, [160].log_data[43].maxminute := 12, [160].log_data[43].valid := 1, [160].log_data[44].min := -0.27999878, [160].log_data[44].max := -0.26000214, [160].log_data[44].total := -939.84174, [160].log_data[44].time := 3600.0, [160].log_data[44].valid := 1, [160].log_data[45].time := 3600.0, [160].log_data[45].valid := 1, [160].log_data[46].time := 3600.0, [160].log_data[46].valid := 1, [160].log_data[47].time := 3600.0, [160].log_data[47].valid := 1, [160].log_data[48].min := 6.673664, [160].log_data[48].max := 6.9152203, [160].log_data[48].total := 24294.744, [160].log_data[48].time := 3600.0, [160].log_data[48].minminute := 57, [160].log_data[48].maxminute := 44, [160].log_data[48].valid := 1, [160].log_data[49].min := 7.5933027, [160].log_data[49].max := 9.471025, [160].log_data[49].total := 31548.71, [160].log_data[49].time := 3600.0,
        [160].log_data[49].maxminute := 42, [160].log_data[49].valid := 1, [160].log_data[50].min := 1.9995611, [160].log_data[50].max := 2.1391244, [160].log_data[50].total := 7500.8486, [160].log_data[50].time := 3600.0, [160].log_data[50].minminute := 31, [160].log_data[50].maxminute := 57, [160].log_data[50].valid := 1, [160].log_data[51].max := 3.1395001, [160].log_data[51].total := 2003.6888, [160].log_data[51].time := 3600.0, [160].log_data[51].maxminute := 12, [160].log_data[51].valid := 1, [160].log_data[52].min := -2.8600006, [160].log_data[52].max := 0.13999939, [160].log_data[52].total := -5652.171, [160].log_data[52].time := 3600.0, [160].log_data[52].minminute := 21, [160].log_data[52].maxminute := 3, [160].log_data[52].valid := 1, [160].log_data[53].min := -2.5800018, [160].log_data[53].max := 0.19999695, [160].log_data[53].total := -5558.679, [160].log_data[53].time := 3600.0, [160].log_data[53].minminute := 13, [160].log_data[53].maxminute := 7, [160].log_data[53].valid := 1, [160].log_data[54].max := 0.5335, [160].log_data[54].total := 528.40796, [160].log_data[54].time := 3600.0, [160].log_data[54].minminute := 2, [160].log_data[54].maxminute := 21, [160].log_data[54].valid := 1, [160].log_data[55].max := 0.5275, [160].log_data[55].total := 551.91156, [160].log_data[55].time := 3600.0, [160].log_data[55].minminute := 2, [160].log_data[55].maxminute := 23, [160].log_data[55].valid := 1, [160].log_data[56].min := 0.16083448, [160].log_data[56].max := 0.16122705, [160].log_data[56].total := 579.5539, [160].log_data[56].time := 3600.0, [160].log_data[56].maxminute := 14, [160].log_data[56].valid := 1, [160].log_data[57].min := 0.3575577, [160].log_data[57].max := 0.35810733, [160].log_data[57].total := 1288.1613, [160].log_data[57].time := 3600.0, [160].log_data[57].maxminute := 40, [160].log_data[57].valid := 1, [160].log_data[58].time := 3600.0, [160].log_data[58].valid := 1, [160].log_data[59].time := 3600.0, [160].log_data[59].valid := 1, [160].log_data[60].valid := 1, [160].log_data[61].valid := 1, [160].log_data[62].valid := 1, [160].log_data[63].valid := 1,
        [160].log_data[64].valid := 1, [160].log_data[65].valid := 1, [160].log_data[66].valid := 1, [160].log_data[67].valid := 1, [160].log_data[68].valid := 1, [160].log_data[69].valid := 1, [160].log_data[70].valid := 1, [160].log_data[71].valid := 1, [160].log_data[72].valid := 1, [160].log_data[73].valid := 1, [160].log_data[74].valid := 1, [160].log_data[75].valid := 1, [160].log_data[76].valid := 1, [160].log_data[77].valid := 1, [160].log_data[78].valid := 1, [160].log_data[79].valid := 1, [160].log_data[80].valid := 1, [160].log_data[81].valid := 1, [160].log_data[82].valid := 1, [160].log_data[83].valid := 1, [160].log_data[84].valid := 1, [160].log_data[85].valid := 1, [160].log_data[86].valid := 1, [160].log_data[87].valid := 1, [160].log_data[88].valid := 1, [160].log_data[89].valid := 1, [160].log_data[90].valid := 1, [160].log_data[91].valid := 1, [160].log_data[92].valid := 1, [160].log_data[93].valid := 1, [160].log_data[94].valid := 1, [160].log_data[95].valid := 1, [160].log_data[96].valid := 1, [160].log_data[97].valid := 1, [160].log_data[98].valid := 1, [160].log_data[99].valid := 1, [160].log_data[100].valid := 1, [160].log_data[101].valid := 1, [160].log_data[102].valid := 1, [160].log_data[103].valid := 1, [160].log_data[104].valid := 1, [160].log_data[105].valid := 1, [160].log_data[106].valid := 1, [160].log_data[107].valid := 1, [160].log_data[108].valid := 1, [160].log_data[109].valid := 1, [160].log_data[110].valid := 1, [160].log_data[111].valid := 1, [160].log_data[112].valid := 1, [160].log_data[113].valid := 1, [160].log_data[114].valid := 1, [160].log_data[115].valid := 1, [160].log_data[116].valid := 1, [160].log_data[117].valid := 1, [160].log_data[118].valid := 1, [160].log_data[119].valid := 1, [160].log_data[120].valid := 1, [160].log_data[121].valid := 1, [160].log_data[122].valid := 1, [160].log_data[123].valid := 1,
        [160].log_data[124].valid := 1, [160].time.Year := 2023, [160].time.Month := 1, [160].time.Day := 11, [160].time.Hour := 11, [160].time.Minute := 59, [160].time.Second := 59, [161].log_data[0].min := 1.0, [161].log_data[0].max := 1.0, [161].log_data[0].total := 3600.0, [161].log_data[0].time := 3600.0, [161].log_data[0].valid := 1, [161].log_data[1].max := 1.0, [161].log_data[1].total := 532.5, [161].log_data[1].time := 3600.0, [161].log_data[1].maxminute := 29, [161].log_data[1].valid := 1, [161].log_data[2].max := 1.0, [161].log_data[2].total := 529.0, [161].log_data[2].time := 3600.0, [161].log_data[2].maxminute := 29, [161].log_data[2].valid := 1, [161].log_data[3].time := 3600.0, [161].log_data[3].valid := 1, [161].log_data[4].time := 3600.0, [161].log_data[4].valid := 1, [161].log_data[5].max := 1.0, [161].log_data[5].total := 231.0, [161].log_data[5].time := 3600.0, [161].log_data[5].maxminute := 32, [161].log_data[5].valid := 1, [161].log_data[6].time := 3600.0, [161].log_data[6].valid := 1, [161].log_data[7].time := 3600.0, [161].log_data[7].valid := 1, [161].log_data[8].max := 1.0, [161].log_data[8].total := 1647.249, [161].log_data[8].time := 3600.0, [161].log_data[8].maxminute := 32, [161].log_data[8].valid := 1, [161].log_data[9].max := 1.0, [161].log_data[9].total := 1643.749, [161].log_data[9].time := 3600.0, [161].log_data[9].maxminute := 32, [161].log_data[9].valid := 1, [161].log_data[10].min := 1.0, [161].log_data[10].max := 1.0, [161].log_data[10].total := 3600.0, [161].log_data[10].time := 3600.0, [161].log_data[10].valid := 1, [161].log_data[11].time := 3600.0, [161].log_data[11].valid := 1, [161].log_data[12].min := 1.0, [161].log_data[12].max := 1.0, [161].log_data[12].total := 3600.0, [161].log_data[12].time := 3600.0, [161].log_data[12].valid := 1, [161].log_data[13].min := 1.0, [161].log_data[13].max := 1.0, [161].log_data[13].total := 3600.0,
        [161].log_data[13].time := 3600.0, [161].log_data[13].valid := 1, [161].log_data[14].time := 3600.0, [161].log_data[14].valid := 1, [161].log_data[15].time := 3600.0, [161].log_data[15].valid := 1, [161].log_data[16].time := 3600.0, [161].log_data[16].valid := 1, [161].log_data[17].min := 1.0, [161].log_data[17].max := 1.0, [161].log_data[17].total := 3600.0, [161].log_data[17].time := 3600.0, [161].log_data[17].valid := 1, [161].log_data[18].time := 3600.0, [161].log_data[18].valid := 1, [161].log_data[19].time := 3600.0, [161].log_data[19].valid := 1, [161].log_data[20].time := 3600.0, [161].log_data[20].valid := 1, [161].log_data[21].min := 1.0, [161].log_data[21].max := 1.0, [161].log_data[21].total := 3600.0, [161].log_data[21].time := 3600.0, [161].log_data[21].valid := 1, [161].log_data[22].time := 3600.0, [161].log_data[22].valid := 1, [161].log_data[23].time := 3600.0, [161].log_data[23].valid := 1, [161].log_data[24].time := 3600.0, [161].log_data[24].valid := 1, [161].log_data[25].time := 3600.0, [161].log_data[25].valid := 1, [161].log_data[26].time := 3600.0, [161].log_data[26].valid := 1, [161].log_data[27].time := 3600.0, [161].log_data[27].valid := 1, [161].log_data[28].time := 3600.0, [161].log_data[28].valid := 1, [161].log_data[29].min := 1.0, [161].log_data[29].max := 1.0, [161].log_data[29].total := 3600.0, [161].log_data[29].time := 3600.0, [161].log_data[29].valid := 1, [161].log_data[30].min := 1.0, [161].log_data[30].max := 1.0, [161].log_data[30].total := 3600.0, [161].log_data[30].time := 3600.0, [161].log_data[30].valid := 1, [161].log_data[31].max := 1.0, [161].log_data[31].total := 543.249, [161].log_data[31].time := 3600.0, [161].log_data[31].maxminute := 43, [161].log_data[31].valid := 1, [161].log_data[32].max := 1.0, [161].log_data[32].total := 920.749, [161].log_data[32].time := 3600.0, [161].log_data[32].maxminute := 32, [161].log_data[32].valid := 1, [161].log_data[33].time := 3600.0, [161].log_data[33].valid := 1,
        [161].log_data[34].time := 3600.0, [161].log_data[34].valid := 1, [161].log_data[35].max := 1.0, [161].log_data[35].total := 752.49805, [161].log_data[35].time := 3600.0, [161].log_data[35].maxminute := 35, [161].log_data[35].valid := 1, [161].log_data[36].max := 1.0, [161].log_data[36].total := 619.498, [161].log_data[36].time := 3600.0, [161].log_data[36].maxminute := 32, [161].log_data[36].valid := 1, [161].log_data[37].max := 7.5037603, [161].log_data[37].total := 3465.921, [161].log_data[37].time := 3600.0, [161].log_data[37].maxminute := 30, [161].log_data[37].valid := 1, [161].log_data[38].time := 3600.0, [161].log_data[38].valid := 1, [161].log_data[39].min := 0.9957663, [161].log_data[39].max := 1.0212055, [161].log_data[39].total := 3608.141, [161].log_data[39].time := 3600.0, [161].log_data[39].minminute := 28, [161].log_data[39].maxminute := 32, [161].log_data[39].valid := 1, [161].log_data[40].min := 7.553049, [161].log_data[40].max := 7.5821795, [161].log_data[40].total := 27242.742, [161].log_data[40].time := 3600.0, [161].log_data[40].minminute := 30, [161].log_data[40].maxminute := 39, [161].log_data[40].valid := 1, [161].log_data[41].min := 0.084764406, [161].log_data[41].max := 0.12991162, [161].log_data[41].total := 369.09885, [161].log_data[41].time := 3600.0, [161].log_data[41].minminute := 51, [161].log_data[41].maxminute := 5, [161].log_data[41].valid := 1, [161].log_data[42].min := 2.2928205, [161].log_data[42].max := 2.2981203, [161].log_data[42].total := 8264.178, [161].log_data[42].time := 3600.0, [161].log_data[42].maxminute := 18, [161].log_data[42].valid := 1, [161].log_data[43].min := -0.26000214, [161].log_data[43].max := -0.23999786, [161].log_data[43].total := -915.0592, [161].log_data[43].time := 3600.0, [161].log_data[43].minminute := 7, [161].log_data[43].valid := 1, [161].log_data[44].min := -0.30000305, [161].log_data[44].max := -0.26000214, [161].log_data[44].total := -1004.88043, [161].log_data[44].time := 3600.0, [161].log_data[44].minminute := 45, [161].log_data[44].valid := 1, [161].log_data[45].time := 3600.0, [161].log_data[45].valid := 1,
        [161].log_data[46].time := 3600.0, [161].log_data[46].valid := 1, [161].log_data[47].time := 3600.0, [161].log_data[47].valid := 1, [161].log_data[48].min := 6.5810537, [161].log_data[48].max := 6.9394035, [161].log_data[48].total := 24139.416, [161].log_data[48].time := 3600.0, [161].log_data[48].minminute := 59, [161].log_data[48].maxminute := 38, [161].log_data[48].valid := 1, [161].log_data[49].min := 6.895683, [161].log_data[49].max := 9.340296, [161].log_data[49].total := 29802.334, [161].log_data[49].time := 3600.0, [161].log_data[49].minminute := 57, [161].log_data[49].maxminute := 32, [161].log_data[49].valid := 1, [161].log_data[50].min := 2.091661, [161].log_data[50].max := 2.1518438, [161].log_data[50].total := 7675.53, [161].log_data[50].time := 3600.0, [161].log_data[50].minminute := 36, [161].log_data[50].maxminute := 32, [161].log_data[50].valid := 1, [161].log_data[51].time := 3600.0, [161].log_data[51].valid := 1, [161].log_data[52].min := -4.079994, [161].log_data[52].max := 0.11999512, [161].log_data[52].total := -6659.4297, [161].log_data[52].time := 3600.0, [161].log_data[52].minminute := 32, [161].log_data[52].maxminute := 41, [161].log_data[52].valid := 1, [161].log_data[53].min := -3.9399948, [161].log_data[53].max := 0.16000366, [161].log_data[53].total := -5936.428, [161].log_data[53].time := 3600.0, [161].log_data[53].minminute := 32, [161].log_data[53].maxminute := 45, [161].log_data[53].valid := 1, [161].log_data[54].max := 0.5165, [161].log_data[54].total := 579.4195, [161].log_data[54].time := 3600.0, [161].log_data[54].maxminute := 43, [161].log_data[54].valid := 1, [161].log_data[55].max := 0.5195, [161].log_data[55].total := 541.0892, [161].log_data[55].time := 3600.0, [161].log_data[55].maxminute := 35, [161].log_data[55].valid := 1, [161].log_data[56].min := 0.16087373, [161].log_data[56].max := 0.16122705, [161].log_data[56].total := 579.64154, [161].log_data[56].time := 3600.0, [161].log_data[56].maxminute := 3, [161].log_data[56].valid := 1, [161].log_data[57].min := 0.3572044, [161].log_data[57].max := 0.35814658, [161].log_data[57].total := 1288.3953,
        [161].log_data[57].time := 3600.0, [161].log_data[57].minminute := 59, [161].log_data[57].maxminute := 24, [161].log_data[57].valid := 1, [161].log_data[58].time := 3600.0, [161].log_data[58].valid := 1, [161].log_data[59].time := 3600.0, [161].log_data[59].valid := 1, [161].log_data[60].valid := 1, [161].log_data[61].valid := 1, [161].log_data[62].valid := 1, [161].log_data[63].valid := 1, [161].log_data[64].valid := 1, [161].log_data[65].valid := 1, [161].log_data[66].valid := 1, [161].log_data[67].valid := 1, [161].log_data[68].valid := 1, [161].log_data[69].valid := 1, [161].log_data[70].valid := 1, [161].log_data[71].valid := 1, [161].log_data[72].valid := 1, [161].log_data[73].valid := 1, [161].log_data[74].valid := 1, [161].log_data[75].valid := 1, [161].log_data[76].valid := 1, [161].log_data[77].valid := 1, [161].log_data[78].valid := 1, [161].log_data[79].valid := 1, [161].log_data[80].valid := 1, [161].log_data[81].valid := 1, [161].log_data[82].valid := 1, [161].log_data[83].valid := 1, [161].log_data[84].valid := 1, [161].log_data[85].valid := 1, [161].log_data[86].valid := 1, [161].log_data[87].valid := 1, [161].log_data[88].valid := 1, [161].log_data[89].valid := 1, [161].log_data[90].valid := 1, [161].log_data[91].valid := 1, [161].log_data[92].valid := 1, [161].log_data[93].valid := 1, [161].log_data[94].valid := 1, [161].log_data[95].valid := 1, [161].log_data[96].valid := 1, [161].log_data[97].valid := 1, [161].log_data[98].valid := 1, [161].log_data[99].valid := 1, [161].log_data[100].valid := 1, [161].log_data[101].valid := 1, [161].log_data[102].valid := 1, [161].log_data[103].valid := 1, [161].log_data[104].valid := 1, [161].log_data[105].valid := 1, [161].log_data[106].valid := 1, [161].log_data[107].valid := 1, [161].log_data[108].valid := 1, [161].log_data[109].valid := 1, [161].log_data[110].valid := 1, [161].log_data[111].valid := 1,
        [161].log_data[112].valid := 1, [161].log_data[113].valid := 1, [161].log_data[114].valid := 1, [161].log_data[115].valid := 1, [161].log_data[116].valid := 1, [161].log_data[117].valid := 1, [161].log_data[118].valid := 1, [161].log_data[119].valid := 1, [161].log_data[120].valid := 1, [161].log_data[121].valid := 1, [161].log_data[122].valid := 1, [161].log_data[123].valid := 1, [161].log_data[124].valid := 1, [161].time.Year := 2023, [161].time.Month := 1, [161].time.Day := 11, [161].time.Hour := 12, [161].time.Minute := 59, [161].time.Second := 59, [162].log_data[0].min := 1.0, [162].log_data[0].max := 1.0, [162].log_data[0].total := 3600.0, [162].log_data[0].time := 3600.0, [162].log_data[0].valid := 1, [162].log_data[1].time := 3600.0, [162].log_data[1].valid := 1, [162].log_data[2].time := 3600.0, [162].log_data[2].valid := 1, [162].log_data[3].time := 3600.0, [162].log_data[3].valid := 1, [162].log_data[4].time := 3600.0, [162].log_data[4].valid := 1, [162].log_data[5].time := 3600.0, [162].log_data[5].valid := 1, [162].log_data[6].time := 3600.0, [162].log_data[6].valid := 1, [162].log_data[7].time := 3600.0, [162].log_data[7].valid := 1, [162].log_data[8].min := 1.0, [162].log_data[8].max := 1.0, [162].log_data[8].total := 3600.0, [162].log_data[8].time := 3600.0, [162].log_data[8].valid := 1, [162].log_data[9].min := 1.0, [162].log_data[9].max := 1.0, [162].log_data[9].total := 3600.0, [162].log_data[9].time := 3600.0, [162].log_data[9].valid := 1, [162].log_data[10].min := 1.0, [162].log_data[10].max := 1.0, [162].log_data[10].total := 3600.0, [162].log_data[10].time := 3600.0, [162].log_data[10].valid := 1, [162].log_data[11].time := 3600.0, [162].log_data[11].valid := 1, [162].log_data[12].min := 1.0, [162].log_data[12].max := 1.0, [162].log_data[12].total := 3600.0, [162].log_data[12].time := 3600.0, [162].log_data[12].valid := 1,
        [162].log_data[13].min := 1.0, [162].log_data[13].max := 1.0, [162].log_data[13].total := 3600.0, [162].log_data[13].time := 3600.0, [162].log_data[13].valid := 1, [162].log_data[14].time := 3600.0, [162].log_data[14].valid := 1, [162].log_data[15].time := 3600.0, [162].log_data[15].valid := 1, [162].log_data[16].time := 3600.0, [162].log_data[16].valid := 1, [162].log_data[17].min := 1.0, [162].log_data[17].max := 1.0, [162].log_data[17].total := 3600.0, [162].log_data[17].time := 3600.0, [162].log_data[17].valid := 1, [162].log_data[18].time := 3600.0, [162].log_data[18].valid := 1, [162].log_data[19].time := 3600.0, [162].log_data[19].valid := 1, [162].log_data[20].time := 3600.0, [162].log_data[20].valid := 1, [162].log_data[21].min := 1.0, [162].log_data[21].max := 1.0, [162].log_data[21].total := 3600.0, [162].log_data[21].time := 3600.0, [162].log_data[21].valid := 1, [162].log_data[22].time := 3600.0, [162].log_data[22].valid := 1, [162].log_data[23].time := 3600.0, [162].log_data[23].valid := 1, [162].log_data[24].time := 3600.0, [162].log_data[24].valid := 1, [162].log_data[25].time := 3600.0, [162].log_data[25].valid := 1, [162].log_data[26].time := 3600.0, [162].log_data[26].valid := 1, [162].log_data[27].time := 3600.0, [162].log_data[27].valid := 1, [162].log_data[28].time := 3600.0, [162].log_data[28].valid := 1, [162].log_data[29].min := 1.0, [162].log_data[29].max := 1.0, [162].log_data[29].total := 3600.0, [162].log_data[29].time := 3600.0, [162].log_data[29].valid := 1, [162].log_data[30].min := 1.0, [162].log_data[30].max := 1.0, [162].log_data[30].total := 3600.0, [162].log_data[30].time := 3600.0, [162].log_data[30].valid := 1, [162].log_data[31].max := 1.0, [162].log_data[31].total := 1629.998, [162].log_data[31].time := 3600.0, [162].log_data[31].maxminute := 4, [162].log_data[31].valid := 1, [162].log_data[32].max := 1.0, [162].log_data[32].total := 1440.7471, [162].log_data[32].time := 3600.0, [162].log_data[32].minminute := 2,
        [162].log_data[32].valid := 1, [162].log_data[33].time := 3600.0, [162].log_data[33].valid := 1, [162].log_data[34].time := 3600.0, [162].log_data[34].valid := 1, [162].log_data[35].max := 1.0, [162].log_data[35].total := 1440.7471, [162].log_data[35].time := 3600.0, [162].log_data[35].minminute := 5, [162].log_data[35].valid := 1, [162].log_data[36].max := 1.0, [162].log_data[36].total := 1629.7471, [162].log_data[36].time := 3600.0, [162].log_data[36].maxminute := 7, [162].log_data[36].valid := 1, [162].log_data[37].time := 3600.0, [162].log_data[37].valid := 1, [162].log_data[38].time := 3600.0, [162].log_data[38].valid := 1, [162].log_data[39].min := 0.99635506, [162].log_data[39].max := 1.005306, [162].log_data[39].total := 3604.8909, [162].log_data[39].time := 3600.0, [162].log_data[39].minminute := 13, [162].log_data[39].maxminute := 22, [162].log_data[39].valid := 1, [162].log_data[40].min := 7.538759, [162].log_data[40].max := 7.586301, [162].log_data[40].total := 27244.49, [162].log_data[40].time := 3600.0, [162].log_data[40].minminute := 47, [162].log_data[40].maxminute := 59, [162].log_data[40].valid := 1, [162].log_data[41].min := 0.0829978, [162].log_data[41].max := 0.14345556, [162].log_data[41].total := 415.8459, [162].log_data[41].time := 3600.0, [162].log_data[41].minminute := 12, [162].log_data[41].maxminute := 28, [162].log_data[41].valid := 1, [162].log_data[42].min := 2.2927027, [162].log_data[42].max := 2.2978847, [162].log_data[42].total := 8264.324, [162].log_data[42].time := 3600.0, [162].log_data[42].minminute := 43, [162].log_data[42].maxminute := 10, [162].log_data[42].valid := 1, [162].log_data[43].min := -0.27999878, [162].log_data[43].max := -0.26000214, [162].log_data[43].total := -937.7937, [162].log_data[43].time := 3600.0, [162].log_data[43].minminute := 32, [162].log_data[43].valid := 1, [162].log_data[44].min := -0.30000305, [162].log_data[44].max := -0.27999878, [162].log_data[44].total := -1059.1074, [162].log_data[44].time := 3600.0, [162].log_data[44].valid := 1, [162].log_data[45].time := 3600.0, [162].log_data[45].valid := 1,
